LIN {X 0,Y 410.932,Z 415.987,A -85,B 0,C 180,E1 -10557.501,E2 -10557.501} C_VEL
LIN {X 0,Y 411.272,Z 410.477,A -85,B 0,C 180,E1 -10560.841,E2 -10560.841} C_VEL
LIN {X 0,Y 411.519,Z 406.698,A -85,B 0,C 180,E1 -10563.193,E2 -10563.193} C_VEL
LIN {X 0,Y 411.867,Z 401.28,A -85,B 0,C 180,E1 -10566.679,E2 -10566.679} C_VEL
LIN {X 0,Y 411.907,Z 397.623,A -85,B 0,C 180,E1 -10569.146,E2 -10569.146} C_VEL
LIN {X 0,Y 411.508,Z 393.953,A -85,B 0,C 180,E1 -10571.764,E2 -10571.764} C_VEL
LIN {X 0,Y 411.201,Z 391.892,A -85,B 0,C 180,E1 -10573.298,E2 -10573.298} C_VEL
LIN {X 0,Y 411.178,Z 391.895,A -85,B 0,C 180,E1 -10576.867,E2 -10576.867} C_VEL
LIN {X 0,Y 411.229,Z 391.886,A -85,B 0,C 180,E1 -10580.27,E2 -10580.27} C_VEL
LIN {X 0,Y 411.197,Z 391.89,A -85,B 0,C 180,E1 -10583.447,E2 -10583.447} C_VEL
LIN {X 0,Y 411.208,Z 391.889,A -85,B 0,C 180,E1 -10586.873,E2 -10586.873} C_VEL
LIN {X 0,Y 411.234,Z 391.888,A -85,B 0,C 180,E1 -10590.644,E2 -10590.644} C_VEL
LIN {X 0,Y 411.238,Z 391.885,A -85,B 0,C 180,E1 -10593.619,E2 -10593.619} C_VEL
LIN {X 0,Y 411.197,Z 391.89,A -85,B 0,C 180,E1 -10596.852,E2 -10596.852} C_VEL
LIN {X 0,Y 411.216,Z 391.887,A -85,B 0,C 180,E1 -10600.05,E2 -10600.05} C_VEL
LIN {X 0,Y 411.266,Z 391.879,A -85,B 0,C 180,E1 -10603.13,E2 -10603.13} C_VEL
LIN {X 0,Y 411.258,Z 391.88,A -85,B 0,C 180,E1 -10606.158,E2 -10606.158} C_VEL
LIN {X 0,Y 411.289,Z 391.876,A -85,B 0,C 180,E1 -10609.166,E2 -10609.166} C_VEL
LIN {X 0,Y 411.483,Z 391.852,A -85,B 0,C 180,E1 -10612.147,E2 -10612.147} C_VEL
LIN {X 0,Y 411.477,Z 391.854,A -85,B 0,C 180,E1 -10614.118,E2 -10614.118} C_VEL
LIN {X 0,Y 411.516,Z 391.85,A -85,B 0,C 180,E1 -10618.043,E2 -10618.043} C_VEL
LIN {X 0,Y 411.644,Z 391.836,A -85,B 0,C 180,E1 -10620,E2 -10620} C_VEL
LIN {X 0,Y 411.459,Z 391.857,A -85,B 0,C 180,E1 -10622.937,E2 -10622.937} C_VEL
LIN {X 0,Y 411.463,Z 391.857,A -85,B 0,C 180,E1 -10626.867,E2 -10626.867} C_VEL
LIN {X 0,Y 411.306,Z 391.878,A -85,B 0,C 180,E1 -10629.839,E2 -10629.839} C_VEL
LIN {X 0,Y 411.307,Z 391.875,A -85,B 0,C 180,E1 -10633.104,E2 -10633.104} C_VEL
LIN {X 0,Y 411.265,Z 391.882,A -85,B 0,C 180,E1 -10635.868,E2 -10635.868} C_VEL
LIN {X 0,Y 411.227,Z 391.885,A -85,B 0,C 180,E1 -10638.949,E2 -10638.949} C_VEL
LIN {X 0,Y 411.206,Z 391.891,A -85,B 0,C 180,E1 -10642.643,E2 -10642.643} C_VEL
LIN {X 0,Y 411.238,Z 391.884,A -85,B 0,C 180,E1 -10645.293,E2 -10645.293} C_VEL
LIN {X 0,Y 411.26,Z 391.884,A -85,B 0,C 180,E1 -10647.478,E2 -10647.478} C_VEL
LIN {X 0,Y 411.191,Z 391.893,A -85,B 0,C 180,E1 -10650.848,E2 -10650.848} C_VEL
LIN {X 0,Y 411.208,Z 391.89,A -85,B 0,C 180,E1 -10654.333,E2 -10654.333} C_VEL
LIN {X 0,Y 411.202,Z 391.887,A -85,B 0,C 180,E1 -10657.973,E2 -10657.973} C_VEL
LIN {X 0,Y 411.183,Z 391.894,A -85,B 0,C 180,E1 -10660.504,E2 -10660.504} C_VEL
LIN {X 0,Y 411.175,Z 391.893,A -85,B 0,C 180,E1 -10663.134,E2 -10663.134} C_VEL
LIN {X 0,Y 411.175,Z 391.894,A -85,B 0,C 180,E1 -10665.88,E2 -10665.88} C_VEL
LIN {X 0,Y 411.196,Z 392.038,A -85,B 0,C 180,E1 -10668.767,E2 -10668.767} C_VEL
LIN {X 0,Y 411.452,Z 394.537,A -85,B 0,C 180,E1 -10670.803,E2 -10670.803} C_VEL
LIN {X 0,Y 411.471,Z 397.876,A -85,B 0,C 180,E1 -10673.396,E2 -10673.396} C_VEL
LIN {X 0,Y 411.254,Z 402.544,A -85,B 0,C 180,E1 -10676.864,E2 -10676.864} C_VEL
LIN {X 0,Y 411.071,Z 405.713,A -85,B 0,C 180,E1 -10679.143,E2 -10679.143} C_VEL
LIN {X 0,Y 410.798,Z 410.981,A -85,B 0,C 180,E1 -10682.827,E2 -10682.827} C_VEL
LIN {X 0,Y 410.582,Z 415.248,A -85,B 0,C 180,E1 -10685.744,E2 -10685.744} C_VEL
LIN {X 0,Y 410.457,Z 419.829,A -85,B 0,C 180,E1 -10688.754,E2 -10688.754} C_VEL
LIN {X 0,Y 414.185,Z 433.819,A -85,B 0,C 180,E1 -10689.343,E2 -10689.343} C_VEL
LIN {X 0,Y 417.104,Z 447.077,A -85,B 0,C 180,E1 -10690.05,E2 -10690.05} C_VEL
LIN {X 0,Y 417.637,Z 450.91,A -85,B 0,C 180,E1 -10690.269,E2 -10690.269} C_VEL
LIN {X 0,Y 416.849,Z 464.097,A -85,B 0,C 180,E1 -10691.04,E2 -10691.04} C_VEL
LIN {X 0,Y 415.977,Z 475.884,A -85,B 0,C 180,E1 -10691.914,E2 -10691.914} C_VEL
LIN {X 0,Y 414.892,Z 487.847,A -85,B 0,C 180,E1 -10693.01,E2 -10693.01} C_VEL
LIN {X 0,Y 413.863,Z 498.759,A -85,B 0,C 180,E1 -10694.234,E2 -10694.234} C_VEL
LIN {X 0,Y 412.988,Z 508.063,A -85,B 0,C 180,E1 -10695.488,E2 -10695.488} C_VEL
LIN {X 0,Y 412.212,Z 517.264,A -85,B 0,C 180,E1 -10696.983,E2 -10696.983} C_VEL
LIN {X 0,Y 411.336,Z 525.8,A -85,B 0,C 180,E1 -10698.669,E2 -10698.669} C_VEL
LIN {X 0,Y 410.849,Z 531.96,A -85,B 0,C 180,E1 -10700.151,E2 -10700.151} C_VEL
LIN {X 0,Y 410.369,Z 538.494,A -85,B 0,C 180,E1 -10702.125,E2 -10702.125} C_VEL
LIN {X 0,Y 410.135,Z 543.392,A -85,B 0,C 180,E1 -10704.099,E2 -10704.099} C_VEL
LIN {X 0,Y 409.939,Z 546.804,A -85,B 0,C 180,E1 -10706.068,E2 -10706.068} C_VEL
LIN {X 0,Y 409.966,Z 548.829,A -85,B 0,C 180,E1 -10708.035,E2 -10708.035} C_VEL
LIN {X 0,Y 409.905,Z 549.526,A -85,B 0,C 180,E1 -10710,E2 -10710} C_VEL
LIN {X 0,Y 409.966,Z 548.9,A -85,B 0,C 180,E1 -10711.965,E2 -10711.965} C_VEL
LIN {X 0,Y 409.938,Z 546.938,A -85,B 0,C 180,E1 -10713.932,E2 -10713.932} C_VEL
LIN {X 0,Y 410.122,Z 543.591,A -85,B 0,C 180,E1 -10715.902,E2 -10715.902} C_VEL
LIN {X 0,Y 410.365,Z 538.765,A -85,B 0,C 180,E1 -10717.875,E2 -10717.875} C_VEL
LIN {X 0,Y 410.488,Z 536.976,A -85,B 0,C 180,E1 -10718.482,E2 -10718.482} C_VEL
LIN {X 0,Y 409.995,Z 534.605,A -85,B 0,C 180,E1 -10719.231,E2 -10719.231} C_VEL
LIN {X 0,Y 407.5,Z 530.401,A -85,B 0,C 180,E1 -10720.443,E2 -10720.443} C_VEL
LIN {X 0,Y 405.098,Z 525.759,A -85,B 0,C 180,E1 -10721.632,E2 -10721.632} C_VEL
LIN {X 0,Y 404.756,Z 522.548,A -85,B 0,C 180,E1 -10722.334,E2 -10722.334} C_VEL
LIN {X 0,Y 405.592,Z 513.315,A -85,B 0,C 180,E1 -10724.04,E2 -10724.04} C_VEL
LIN {X 0,Y 406.577,Z 503.364,A -85,B 0,C 180,E1 -10725.541,E2 -10725.541} C_VEL
LIN {X 0,Y 407.689,Z 492.287,A -85,B 0,C 180,E1 -10726.912,E2 -10726.912} C_VEL
LIN {X 0,Y 408.768,Z 481.257,A -85,B 0,C 180,E1 -10728.028,E2 -10728.028} C_VEL
LIN {X 0,Y 409.79,Z 469.285,A -85,B 0,C 180,E1 -10729.018,E2 -10729.018} C_VEL
LIN {X 0,Y 410.684,Z 456.556,A -85,B 0,C 180,E1 -10729.855,E2 -10729.855} C_VEL
LIN {X 0,Y 410.884,Z 450.89,A -85,B 0,C 180,E1 -10730.172,E2 -10730.172} C_VEL
LIN {X 0,Y 407.936,Z 436.771,A -85,B 0,C 180,E1 -10730.982,E2 -10730.982} C_VEL
LIN {X 0,Y 404.018,Z 422.414,A -85,B 0,C 180,E1 -10731.644,E2 -10731.644} C_VEL
LIN {X 0,Y 403.384,Z 419.805,A -85,B 0,C 180,E1 -10731.747,E2 -10731.747} C_VEL
LIN {X 0,Y 403.588,Z 414.887,A -85,B 0,C 180,E1 -10735.107,E2 -10735.107} C_VEL
LIN {X 0,Y 403.764,Z 410.679,A -85,B 0,C 180,E1 -10738.032,E2 -10738.032} C_VEL
LIN {X 0,Y 404.09,Z 405.774,A -85,B 0,C 180,E1 -10741.546,E2 -10741.546} C_VEL
LIN {X 0,Y 404.322,Z 401.114,A -85,B 0,C 180,E1 -10745.003,E2 -10745.003} C_VEL
LIN {X 0,Y 404.462,Z 397.921,A -85,B 0,C 180,E1 -10747.457,E2 -10747.457} C_VEL
LIN {X 0,Y 404.367,Z 394.599,A -85,B 0,C 180,E1 -10750.117,E2 -10750.117} C_VEL
LIN {X 0,Y 404.167,Z 392.814,A -85,B 0,C 180,E1 -10751.606,E2 -10751.606} C_VEL
LIN {X 0,Y 404.151,Z 392.773,A -85,B 0,C 180,E1 -10754.523,E2 -10754.523} C_VEL
LIN {X 0,Y 404.139,Z 392.772,A -85,B 0,C 180,E1 -10757.296,E2 -10757.296} C_VEL
LIN {X 0,Y 404.171,Z 392.766,A -85,B 0,C 180,E1 -10759.955,E2 -10759.955} C_VEL
LIN {X 0,Y 404.143,Z 392.769,A -85,B 0,C 180,E1 -10763.124,E2 -10763.124} C_VEL
LIN {X 0,Y 404.148,Z 392.77,A -85,B 0,C 180,E1 -10766.188,E2 -10766.188} C_VEL
LIN {X 0,Y 404.148,Z 392.767,A -85,B 0,C 180,E1 -10769.715,E2 -10769.715} C_VEL
LIN {X 0,Y 404.198,Z 392.761,A -85,B 0,C 180,E1 -10773.123,E2 -10773.123} C_VEL
LIN {X 0,Y 404.18,Z 392.764,A -85,B 0,C 180,E1 -10775.334,E2 -10775.334} C_VEL
LIN {X 0,Y 404.142,Z 392.769,A -85,B 0,C 180,E1 -10778.581,E2 -10778.581} C_VEL
LIN {X 0,Y 404.213,Z 392.76,A -85,B 0,C 180,E1 -10781.762,E2 -10781.762} C_VEL
LIN {X 0,Y 404.21,Z 392.759,A -85,B 0,C 180,E1 -10784.882,E2 -10784.882} C_VEL
LIN {X 0,Y 404.26,Z 392.753,A -85,B 0,C 180,E1 -10787.958,E2 -10787.958} C_VEL
LIN {X 0,Y 404.436,Z 392.734,A -85,B 0,C 180,E1 -10792.1,E2 -10792.1} C_VEL
LIN {X 0,Y 404.427,Z 392.733,A -85,B 0,C 180,E1 -10794.015,E2 -10794.015} C_VEL
LIN {X 0,Y 404.483,Z 392.726,A -85,B 0,C 180,E1 -10798.008,E2 -10798.008} C_VEL
LIN {X 0,Y 404.613,Z 392.713,A -85,B 0,C 180,E1 -10800,E2 -10800} C_VEL
LIN {X 0,Y 404.425,Z 392.734,A -85,B 0,C 180,E1 -10802.988,E2 -10802.988} C_VEL
LIN {X 0,Y 404.415,Z 392.734,A -85,B 0,C 180,E1 -10806.987,E2 -10806.987} C_VEL
LIN {X 0,Y 404.269,Z 392.753,A -85,B 0,C 180,E1 -10810.011,E2 -10810.011} C_VEL
LIN {X 0,Y 404.269,Z 392.755,A -85,B 0,C 180,E1 -10813.211,E2 -10813.211} C_VEL
LIN {X 0,Y 404.218,Z 392.757,A -85,B 0,C 180,E1 -10817.007,E2 -10817.007} C_VEL
LIN {X 0,Y 404.166,Z 392.765,A -85,B 0,C 180,E1 -10820.351,E2 -10820.351} C_VEL
LIN {X 0,Y 404.172,Z 392.761,A -85,B 0,C 180,E1 -10823.574,E2 -10823.574} C_VEL
LIN {X 0,Y 404.186,Z 392.764,A -85,B 0,C 180,E1 -10825.766,E2 -10825.766} C_VEL
LIN {X 0,Y 404.197,Z 392.762,A -85,B 0,C 180,E1 -10827.999,E2 -10827.999} C_VEL
LIN {X 0,Y 404.141,Z 392.768,A -85,B 0,C 180,E1 -10831.558,E2 -10831.558} C_VEL
LIN {X 0,Y 404.188,Z 392.763,A -85,B 0,C 180,E1 -10835.016,E2 -10835.016} C_VEL
LIN {X 0,Y 404.166,Z 392.77,A -85,B 0,C 180,E1 -10838.756,E2 -10838.756} C_VEL
LIN {X 0,Y 404.152,Z 392.77,A -85,B 0,C 180,E1 -10841.604,E2 -10841.604} C_VEL
LIN {X 0,Y 404.147,Z 392.769,A -85,B 0,C 180,E1 -10844.522,E2 -10844.522} C_VEL
LIN {X 0,Y 404.136,Z 392.807,A -85,B 0,C 180,E1 -10846.454,E2 -10846.454} C_VEL
LIN {X 0,Y 404.641,Z 395.775,A -85,B 0,C 180,E1 -10848.7,E2 -10848.7} C_VEL
LIN {X 0,Y 404.907,Z 399.477,A -85,B 0,C 180,E1 -10851.359,E2 -10851.359} C_VEL
LIN {X 0,Y 404.78,Z 403.102,A -85,B 0,C 180,E1 -10853.82,E2 -10853.82} C_VEL
LIN {X 0,Y 404.389,Z 408.592,A -85,B 0,C 180,E1 -10857.401,E2 -10857.401} C_VEL
LIN {X 0,Y 404.057,Z 414.115,A -85,B 0,C 180,E1 -10860.855,E2 -10860.855} C_VEL
LIN {X 0,Y 403.843,Z 417.797,A -85,B 0,C 180,E1 -10863.097,E2 -10863.097} C_VEL
LIN {X 0,Y 403.539,Z 423.318,A -85,B 0,C 180,E1 -10866.386,E2 -10866.386} C_VEL
LIN {X 0,Y 403.447,Z 426.603,A -85,B 0,C 180,E1 -10868.3,E2 -10868.3} C_VEL
LIN {X 0,Y 407.112,Z 441.134,A -85,B 0,C 180,E1 -10868.91,E2 -10868.91} C_VEL
LIN {X 0,Y 409.79,Z 453.958,A -85,B 0,C 180,E1 -10869.593,E2 -10869.593} C_VEL
LIN {X 0,Y 410.664,Z 460.503,A -85,B 0,C 180,E1 -10869.984,E2 -10869.984} C_VEL
LIN {X 0,Y 409.806,Z 474.005,A -85,B 0,C 180,E1 -10870.822,E2 -10870.822} C_VEL
LIN {X 0,Y 408.723,Z 486.899,A -85,B 0,C 180,E1 -10871.841,E2 -10871.841} C_VEL
LIN {X 0,Y 407.496,Z 499.461,A -85,B 0,C 180,E1 -10873.08,E2 -10873.08} C_VEL
LIN {X 0,Y 406.404,Z 510.651,A -85,B 0,C 180,E1 -10874.452,E2 -10874.452} C_VEL
LIN {X 0,Y 405.407,Z 520.686,A -85,B 0,C 180,E1 -10875.954,E2 -10875.954} C_VEL
LIN {X 0,Y 404.707,Z 529.022,A -85,B 0,C 180,E1 -10877.463,E2 -10877.463} C_VEL
LIN {X 0,Y 403.888,Z 536.989,A -85,B 0,C 180,E1 -10879.219,E2 -10879.219} C_VEL
LIN {X 0,Y 403.433,Z 543.405,A -85,B 0,C 180,E1 -10880.98,E2 -10880.98} C_VEL
LIN {X 0,Y 403.072,Z 549.091,A -85,B 0,C 180,E1 -10882.989,E2 -10882.989} C_VEL
LIN {X 0,Y 402.914,Z 553.217,A -85,B 0,C 180,E1 -10884.997,E2 -10884.997} C_VEL
LIN {X 0,Y 402.779,Z 555.911,A -85,B 0,C 180,E1 -10886.999,E2 -10886.999} C_VEL
LIN {X 0,Y 402.843,Z 557.247,A -85,B 0,C 180,E1 -10889,E2 -10889} C_VEL
LIN {X 0,Y 402.843,Z 557.246,A -85,B 0,C 180,E1 -10891,E2 -10891} C_VEL
LIN {X 0,Y 402.779,Z 555.909,A -85,B 0,C 180,E1 -10893.001,E2 -10893.001} C_VEL
LIN {X 0,Y 402.918,Z 553.214,A -85,B 0,C 180,E1 -10895.003,E2 -10895.003} C_VEL
LIN {X 0,Y 403.077,Z 549.081,A -85,B 0,C 180,E1 -10897.01,E2 -10897.01} C_VEL
LIN {X 0,Y 403.418,Z 543.388,A -85,B 0,C 180,E1 -10899.021,E2 -10899.021} C_VEL
LIN {X 0,Y 403.888,Z 536.97,A -85,B 0,C 180,E1 -10900.781,E2 -10900.781} C_VEL
LIN {X 0,Y 404.707,Z 528.998,A -85,B 0,C 180,E1 -10902.537,E2 -10902.537} C_VEL
LIN {X 0,Y 405.409,Z 520.656,A -85,B 0,C 180,E1 -10904.046,E2 -10904.046} C_VEL
LIN {X 0,Y 406.395,Z 510.613,A -85,B 0,C 180,E1 -10905.548,E2 -10905.548} C_VEL
LIN {X 0,Y 407.534,Z 499.41,A -85,B 0,C 180,E1 -10906.919,E2 -10906.919} C_VEL
LIN {X 0,Y 408.742,Z 486.838,A -85,B 0,C 180,E1 -10908.158,E2 -10908.158} C_VEL
LIN {X 0,Y 409.746,Z 474.198,A -85,B 0,C 180,E1 -10909.161,E2 -10909.161} C_VEL
LIN {X 0,Y 410.658,Z 460.385,A -85,B 0,C 180,E1 -10910.016,E2 -10910.016} C_VEL
LIN {X 0,Y 408.735,Z 448.556,A -85,B 0,C 180,E1 -10910.704,E2 -10910.704} C_VEL
LIN {X 0,Y 405.445,Z 434.421,A -85,B 0,C 180,E1 -10911.388,E2 -10911.388} C_VEL
LIN {X 0,Y 403.425,Z 426.53,A -85,B 0,C 180,E1 -10911.727,E2 -10911.727} C_VEL
LIN {X 0,Y 403.646,Z 420.745,A -85,B 0,C 180,E1 -10915.125,E2 -10915.125} C_VEL
LIN {X 0,Y 403.928,Z 415.947,A -85,B 0,C 180,E1 -10918.02,E2 -10918.02} C_VEL
LIN {X 0,Y 404.295,Z 410.171,A -85,B 0,C 180,E1 -10921.594,E2 -10921.594} C_VEL
LIN {X 0,Y 404.632,Z 404.91,A -85,B 0,C 180,E1 -10924.972,E2 -10924.972} C_VEL
LIN {X 0,Y 404.882,Z 401.238,A -85,B 0,C 180,E1 -10927.411,E2 -10927.411} C_VEL
LIN {X 0,Y 404.82,Z 397.26,A -85,B 0,C 180,E1 -10930.193,E2 -10930.193} C_VEL
LIN {X 0,Y 404.258,Z 393.357,A -85,B 0,C 180,E1 -10933.1,E2 -10933.1} C_VEL
LIN {X 0,Y 404.135,Z 392.772,A -85,B 0,C 180,E1 -10933.678,E2 -10933.678} C_VEL
LIN {X 0,Y 404.172,Z 392.768,A -85,B 0,C 180,E1 -10937.3,E2 -10937.3} C_VEL
LIN {X 0,Y 404.169,Z 392.767,A -85,B 0,C 180,E1 -10939.955,E2 -10939.955} C_VEL
LIN {X 0,Y 404.142,Z 392.77,A -85,B 0,C 180,E1 -10943.124,E2 -10943.124} C_VEL
LIN {X 0,Y 404.146,Z 392.771,A -85,B 0,C 180,E1 -10946.188,E2 -10946.188} C_VEL
LIN {X 0,Y 404.146,Z 392.769,A -85,B 0,C 180,E1 -10949.715,E2 -10949.715} C_VEL
LIN {X 0,Y 404.196,Z 392.761,A -85,B 0,C 180,E1 -10953.123,E2 -10953.123} C_VEL
LIN {X 0,Y 404.175,Z 392.765,A -85,B 0,C 180,E1 -10955.334,E2 -10955.334} C_VEL
LIN {X 0,Y 404.139,Z 392.769,A -85,B 0,C 180,E1 -10958.581,E2 -10958.581} C_VEL
LIN {X 0,Y 404.212,Z 392.759,A -85,B 0,C 180,E1 -10961.762,E2 -10961.762} C_VEL
LIN {X 0,Y 404.214,Z 392.759,A -85,B 0,C 180,E1 -10964.882,E2 -10964.882} C_VEL
LIN {X 0,Y 404.258,Z 392.753,A -85,B 0,C 180,E1 -10967.959,E2 -10967.959} C_VEL
LIN {X 0,Y 404.435,Z 392.73,A -85,B 0,C 180,E1 -10972.1,E2 -10972.1} C_VEL
LIN {X 0,Y 404.426,Z 392.733,A -85,B 0,C 180,E1 -10974.015,E2 -10974.015} C_VEL
LIN {X 0,Y 404.485,Z 392.726,A -85,B 0,C 180,E1 -10978.009,E2 -10978.009} C_VEL
LIN {X 0,Y 404.613,Z 392.712,A -85,B 0,C 180,E1 -10980,E2 -10980} C_VEL
LIN {X 0,Y 404.418,Z 392.734,A -85,B 0,C 180,E1 -10982.989,E2 -10982.989} C_VEL
LIN {X 0,Y 404.414,Z 392.734,A -85,B 0,C 180,E1 -10986.987,E2 -10986.987} C_VEL
LIN {X 0,Y 404.268,Z 392.753,A -85,B 0,C 180,E1 -10990.012,E2 -10990.012} C_VEL
LIN {X 0,Y 404.268,Z 392.751,A -85,B 0,C 180,E1 -10993.211,E2 -10993.211} C_VEL
LIN {X 0,Y 404.221,Z 392.755,A -85,B 0,C 180,E1 -10997.009,E2 -10997.009} C_VEL
LIN {X 0,Y 404.165,Z 392.764,A -85,B 0,C 180,E1 -11000.352,E2 -11000.352} C_VEL
LIN {X 0,Y 404.171,Z 392.764,A -85,B 0,C 180,E1 -11003.575,E2 -11003.575} C_VEL
LIN {X 0,Y 404.185,Z 392.765,A -85,B 0,C 180,E1 -11005.766,E2 -11005.766} C_VEL
LIN {X 0,Y 404.197,Z 392.762,A -85,B 0,C 180,E1 -11008,E2 -11008} C_VEL
LIN {X 0,Y 404.14,Z 392.768,A -85,B 0,C 180,E1 -11011.558,E2 -11011.558} C_VEL
LIN {X 0,Y 404.187,Z 392.762,A -85,B 0,C 180,E1 -11015.016,E2 -11015.016} C_VEL
LIN {X 0,Y 404.16,Z 392.767,A -85,B 0,C 180,E1 -11018.757,E2 -11018.757} C_VEL
LIN {X 0,Y 404.124,Z 392.77,A -85,B 0,C 180,E1 -11021.6,E2 -11021.6} C_VEL
LIN {X 0,Y 404.148,Z 392.768,A -85,B 0,C 180,E1 -11024.522,E2 -11024.522} C_VEL
LIN {X 0,Y 404.142,Z 392.771,A -85,B 0,C 180,E1 -11027.296,E2 -11027.296} C_VEL
LIN {X 0,Y 404.16,Z 392.979,A -85,B 0,C 180,E1 -11028.64,E2 -11028.64} C_VEL
LIN {X 0,Y 404.451,Z 396.387,A -85,B 0,C 180,E1 -11031.44,E2 -11031.44} C_VEL
LIN {X 0,Y 404.391,Z 399.375,A -85,B 0,C 180,E1 -11033.78,E2 -11033.78} C_VEL
LIN {X 0,Y 404.218,Z 403.085,A -85,B 0,C 180,E1 -11036.57,E2 -11036.57} C_VEL
LIN {X 0,Y 403.939,Z 407.362,A -85,B 0,C 180,E1 -11039.698,E2 -11039.698} C_VEL
LIN {X 0,Y 403.73,Z 412.128,A -85,B 0,C 180,E1 -11043.089,E2 -11043.089} C_VEL
LIN {X 0,Y 403.48,Z 416.909,A -85,B 0,C 180,E1 -11046.383,E2 -11046.383} C_VEL
LIN {X 0,Y 403.416,Z 419.809,A -85,B 0,C 180,E1 -11048.356,E2 -11048.356} C_VEL
LIN {X 0,Y 407.494,Z 435.085,A -85,B 0,C 180,E1 -11049.031,E2 -11049.031} C_VEL
LIN {X 0,Y 410.403,Z 448.443,A -85,B 0,C 180,E1 -11049.775,E2 -11049.775} C_VEL
LIN {X 0,Y 410.898,Z 452.117,A -85,B 0,C 180,E1 -11049.996,E2 -11049.996} C_VEL
LIN {X 0,Y 410.111,Z 464.554,A -85,B 0,C 180,E1 -11050.745,E2 -11050.745} C_VEL
LIN {X 0,Y 409.097,Z 477.382,A -85,B 0,C 180,E1 -11051.728,E2 -11051.728} C_VEL
LIN {X 0,Y 407.826,Z 490.264,A -85,B 0,C 180,E1 -11052.965,E2 -11052.965} C_VEL
LIN {X 0,Y 406.808,Z 500.78,A -85,B 0,C 180,E1 -11054.211,E2 -11054.211} C_VEL
LIN {X 0,Y 405.763,Z 511.22,A -85,B 0,C 180,E1 -11055.711,E2 -11055.711} C_VEL
LIN {X 0,Y 405.038,Z 519.829,A -85,B 0,C 180,E1 -11057.219,E2 -11057.219} C_VEL
LIN {X 0,Y 404.144,Z 528.084,A -85,B 0,C 180,E1 -11058.972,E2 -11058.972} C_VEL
LIN {X 0,Y 403.669,Z 533.835,A -85,B 0,C 180,E1 -11060.48,E2 -11060.48} C_VEL
LIN {X 0,Y 403.309,Z 538.564,A -85,B 0,C 180,E1 -11061.987,E2 -11061.987} C_VEL
LIN {X 0,Y 403.061,Z 543.462,A -85,B 0,C 180,E1 -11063.995,E2 -11063.995} C_VEL
LIN {X 0,Y 402.862,Z 546.873,A -85,B 0,C 180,E1 -11065.999,E2 -11065.999} C_VEL
LIN {X 0,Y 402.864,Z 548.899,A -85,B 0,C 180,E1 -11068.001,E2 -11068.001} C_VEL
LIN {X 0,Y 402.831,Z 549.595,A -85,B 0,C 180,E1 -11070,E2 -11070} C_VEL
LIN {X 0,Y 402.863,Z 548.968,A -85,B 0,C 180,E1 -11072,E2 -11072} C_VEL
LIN {X 0,Y 402.861,Z 547.006,A -85,B 0,C 180,E1 -11074.002,E2 -11074.002} C_VEL
LIN {X 0,Y 403.066,Z 543.659,A -85,B 0,C 180,E1 -11076.005,E2 -11076.005} C_VEL
LIN {X 0,Y 403.305,Z 538.833,A -85,B 0,C 180,E1 -11078.014,E2 -11078.014} C_VEL
LIN {X 0,Y 403.812,Z 532.37,A -85,B 0,C 180,E1 -11080.023,E2 -11080.023} C_VEL
LIN {X 0,Y 404.482,Z 525.173,A -85,B 0,C 180,E1 -11081.78,E2 -11081.78} C_VEL
LIN {X 0,Y 404.756,Z 522.548,A -85,B 0,C 180,E1 -11082.334,E2 -11082.334} C_VEL
LIN {X 0,Y 404.417,Z 519.204,A -85,B 0,C 180,E1 -11083.022,E2 -11083.022} C_VEL
LIN {X 0,Y 402.101,Z 513.578,A -85,B 0,C 180,E1 -11084.14,E2 -11084.14} C_VEL
LIN {X 0,Y 399.893,Z 507.491,A -85,B 0,C 180,E1 -11085.213,E2 -11085.213} C_VEL
LIN {X 0,Y 399.716,Z 503.39,A -85,B 0,C 180,E1 -11085.821,E2 -11085.821} C_VEL
LIN {X 0,Y 400.882,Z 492.352,A -85,B 0,C 180,E1 -11087.208,E2 -11087.208} C_VEL
LIN {X 0,Y 402.01,Z 481.321,A -85,B 0,C 180,E1 -11088.342,E2 -11088.342} C_VEL
LIN {X 0,Y 403.143,Z 468.201,A -85,B 0,C 180,E1 -11089.43,E2 -11089.43} C_VEL
LIN {X 0,Y 404.062,Z 455.371,A -85,B 0,C 180,E1 -11090.268,E2 -11090.268} C_VEL
LIN {X 0,Y 404.018,Z 451.377,A -85,B 0,C 180,E1 -11090.506,E2 -11090.506} C_VEL
LIN {X 0,Y 401.064,Z 437.305,A -85,B 0,C 180,E1 -11091.341,E2 -11091.341} C_VEL
LIN {X 0,Y 397.142,Z 422.944,A -85,B 0,C 180,E1 -11092.027,E2 -11092.027} C_VEL
LIN {X 0,Y 396.32,Z 419.873,A -85,B 0,C 180,E1 -11092.158,E2 -11092.158} C_VEL
LIN {X 0,Y 396.549,Z 415.296,A -85,B 0,C 180,E1 -11095.328,E2 -11095.328} C_VEL
LIN {X 0,Y 396.739,Z 410.746,A -85,B 0,C 180,E1 -11098.574,E2 -11098.574} C_VEL
LIN {X 0,Y 397.06,Z 405.967,A -85,B 0,C 180,E1 -11102.073,E2 -11102.073} C_VEL
LIN {X 0,Y 397.316,Z 401.388,A -85,B 0,C 180,E1 -11105.543,E2 -11105.543} C_VEL
LIN {X 0,Y 397.436,Z 397.971,A -85,B 0,C 180,E1 -11108.237,E2 -11108.237} C_VEL
LIN {X 0,Y 397.251,Z 394.759,A -85,B 0,C 180,E1 -11110.889,E2 -11110.889} C_VEL
LIN {X 0,Y 397.105,Z 393.648,A -85,B 0,C 180,E1 -11111.985,E2 -11111.985} C_VEL
LIN {X 0,Y 397.092,Z 393.649,A -85,B 0,C 180,E1 -11115.068,E2 -11115.068} C_VEL
LIN {X 0,Y 397.069,Z 393.654,A -85,B 0,C 180,E1 -11118.021,E2 -11118.021} C_VEL
LIN {X 0,Y 397.135,Z 393.644,A -85,B 0,C 180,E1 -11121.138,E2 -11121.138} C_VEL
LIN {X 0,Y 397.123,Z 393.646,A -85,B 0,C 180,E1 -11124.496,E2 -11124.496} C_VEL
LIN {X 0,Y 397.081,Z 393.648,A -85,B 0,C 180,E1 -11127.928,E2 -11127.928} C_VEL
LIN {X 0,Y 397.125,Z 393.642,A -85,B 0,C 180,E1 -11131.456,E2 -11131.456} C_VEL
LIN {X 0,Y 397.156,Z 393.639,A -85,B 0,C 180,E1 -11134.488,E2 -11134.488} C_VEL
LIN {X 0,Y 397.112,Z 393.643,A -85,B 0,C 180,E1 -11137.086,E2 -11137.086} C_VEL
LIN {X 0,Y 397.151,Z 393.637,A -85,B 0,C 180,E1 -11140.353,E2 -11140.353} C_VEL
LIN {X 0,Y 397.17,Z 393.638,A -85,B 0,C 180,E1 -11143.553,E2 -11143.553} C_VEL
LIN {X 0,Y 397.231,Z 393.629,A -85,B 0,C 180,E1 -11146.703,E2 -11146.703} C_VEL
LIN {X 0,Y 397.221,Z 393.63,A -85,B 0,C 180,E1 -11149.809,E2 -11149.809} C_VEL
LIN {X 0,Y 397.367,Z 393.611,A -85,B 0,C 180,E1 -11152.888,E2 -11152.888} C_VEL
LIN {X 0,Y 397.257,Z 393.627,A -85,B 0,C 180,E1 -11154.925,E2 -11154.925} C_VEL
LIN {X 0,Y 397.452,Z 393.602,A -85,B 0,C 180,E1 -11157.973,E2 -11157.973} C_VEL
LIN {X 0,Y 397.582,Z 393.588,A -85,B 0,C 180,E1 -11160,E2 -11160} C_VEL
LIN {X 0,Y 397.384,Z 393.612,A -85,B 0,C 180,E1 -11163.041,E2 -11163.041} C_VEL
LIN {X 0,Y 397.367,Z 393.612,A -85,B 0,C 180,E1 -11167.112,E2 -11167.112} C_VEL
LIN {X 0,Y 397.227,Z 393.629,A -85,B 0,C 180,E1 -11170.191,E2 -11170.191} C_VEL
LIN {X 0,Y 397.229,Z 393.631,A -85,B 0,C 180,E1 -11173.321,E2 -11173.321} C_VEL
LIN {X 0,Y 397.184,Z 393.633,A -85,B 0,C 180,E1 -11177.155,E2 -11177.155} C_VEL
LIN {X 0,Y 397.105,Z 393.646,A -85,B 0,C 180,E1 -11180.73,E2 -11180.73} C_VEL
LIN {X 0,Y 397.136,Z 393.638,A -85,B 0,C 180,E1 -11184.018,E2 -11184.018} C_VEL
LIN {X 0,Y 397.196,Z 393.632,A -85,B 0,C 180,E1 -11187.39,E2 -11187.39} C_VEL
LIN {X 0,Y 397.081,Z 393.65,A -85,B 0,C 180,E1 -11190.882,E2 -11190.882} C_VEL
LIN {X 0,Y 397.128,Z 393.644,A -85,B 0,C 180,E1 -11194.493,E2 -11194.493} C_VEL
LIN {X 0,Y 397.112,Z 393.647,A -85,B 0,C 180,E1 -11198.274,E2 -11198.274} C_VEL
LIN {X 0,Y 397.115,Z 393.647,A -85,B 0,C 180,E1 -11200.905,E2 -11200.905} C_VEL
LIN {X 0,Y 397.104,Z 393.648,A -85,B 0,C 180,E1 -11203.648,E2 -11203.648} C_VEL
LIN {X 0,Y 397.108,Z 393.668,A -85,B 0,C 180,E1 -11206.177,E2 -11206.177} C_VEL
LIN {X 0,Y 397.693,Z 397.56,A -85,B 0,C 180,E1 -11209.166,E2 -11209.166} C_VEL
LIN {X 0,Y 397.871,Z 401.218,A -85,B 0,C 180,E1 -11211.812,E2 -11211.812} C_VEL
LIN {X 0,Y 397.685,Z 404.966,A -85,B 0,C 180,E1 -11214.383,E2 -11214.383} C_VEL
LIN {X 0,Y 397.294,Z 410.374,A -85,B 0,C 180,E1 -11217.948,E2 -11217.948} C_VEL
LIN {X 0,Y 396.931,Z 415.89,A -85,B 0,C 180,E1 -11221.441,E2 -11221.441} C_VEL
LIN {X 0,Y 396.608,Z 421.131,A -85,B 0,C 180,E1 -11224.653,E2 -11224.653} C_VEL
LIN {X 0,Y 396.394,Z 426.516,A -85,B 0,C 180,E1 -11227.892,E2 -11227.892} C_VEL
LIN {X 0,Y 400.219,Z 441.498,A -85,B 0,C 180,E1 -11228.544,E2 -11228.544} C_VEL
LIN {X 0,Y 403.125,Z 455.373,A -85,B 0,C 180,E1 -11229.316,E2 -11229.316} C_VEL
LIN {X 0,Y 403.905,Z 460.439,A -85,B 0,C 180,E1 -11229.635,E2 -11229.635} C_VEL
LIN {X 0,Y 403.22,Z 472.633,A -85,B 0,C 180,E1 -11230.398,E2 -11230.398} C_VEL
LIN {X 0,Y 402.068,Z 485.407,A -85,B 0,C 180,E1 -11231.397,E2 -11231.397} C_VEL
LIN {X 0,Y 400.919,Z 497.047,A -85,B 0,C 180,E1 -11232.53,E2 -11232.53} C_VEL
LIN {X 0,Y 399.938,Z 506.736,A -85,B 0,C 180,E1 -11233.67,E2 -11233.67} C_VEL
LIN {X 0,Y 398.777,Z 517.469,A -85,B 0,C 180,E1 -11235.194,E2 -11235.194} C_VEL
LIN {X 0,Y 397.905,Z 526.332,A -85,B 0,C 180,E1 -11236.726,E2 -11236.726} C_VEL
LIN {X 0,Y 397.254,Z 533.707,A -85,B 0,C 180,E1 -11238.261,E2 -11238.261} C_VEL
LIN {X 0,Y 396.679,Z 539.855,A -85,B 0,C 180,E1 -11239.795,E2 -11239.795} C_VEL
LIN {X 0,Y 396.15,Z 546.385,A -85,B 0,C 180,E1 -11241.841,E2 -11241.841} C_VEL
LIN {X 0,Y 395.909,Z 551.272,A -85,B 0,C 180,E1 -11243.886,E2 -11243.886} C_VEL
LIN {X 0,Y 395.754,Z 554.669,A -85,B 0,C 180,E1 -11245.927,E2 -11245.927} C_VEL
LIN {X 0,Y 395.717,Z 556.678,A -85,B 0,C 180,E1 -11247.964,E2 -11247.964} C_VEL
LIN {X 0,Y 395.758,Z 557.344,A -85,B 0,C 180,E1 -11250,E2 -11250} C_VEL
LIN {X 0,Y 395.717,Z 556.676,A -85,B 0,C 180,E1 -11252.035,E2 -11252.035} C_VEL
LIN {X 0,Y 395.755,Z 554.666,A -85,B 0,C 180,E1 -11254.073,E2 -11254.073} C_VEL
LIN {X 0,Y 395.909,Z 551.264,A -85,B 0,C 180,E1 -11256.114,E2 -11256.114} C_VEL
LIN {X 0,Y 396.15,Z 546.368,A -85,B 0,C 180,E1 -11258.159,E2 -11258.159} C_VEL
LIN {X 0,Y 396.678,Z 539.835,A -85,B 0,C 180,E1 -11260.205,E2 -11260.205} C_VEL
LIN {X 0,Y 397.343,Z 532.565,A -85,B 0,C 180,E1 -11261.995,E2 -11261.995} C_VEL
LIN {X 0,Y 398.165,Z 523.994,A -85,B 0,C 180,E1 -11263.707,E2 -11263.707} C_VEL
LIN {X 0,Y 399.133,Z 514.109,A -85,B 0,C 180,E1 -11265.315,E2 -11265.315} C_VEL
LIN {X 0,Y 400.247,Z 503.647,A -85,B 0,C 180,E1 -11266.71,E2 -11266.71} C_VEL
LIN {X 0,Y 401.432,Z 492.101,A -85,B 0,C 180,E1 -11267.973,E2 -11267.973} C_VEL
LIN {X 0,Y 402.622,Z 479.291,A -85,B 0,C 180,E1 -11269.104,E2 -11269.104} C_VEL
LIN {X 0,Y 403.69,Z 465.532,A -85,B 0,C 180,E1 -11270.061,E2 -11270.061} C_VEL
LIN {X 0,Y 403.706,Z 459.176,A -85,B 0,C 180,E1 -11270.442,E2 -11270.442} C_VEL
LIN {X 0,Y 401.095,Z 445.237,A -85,B 0,C 180,E1 -11271.259,E2 -11271.259} C_VEL
LIN {X 0,Y 397.531,Z 431.021,A -85,B 0,C 180,E1 -11271.93,E2 -11271.93} C_VEL
LIN {X 0,Y 396.372,Z 426.475,A -85,B 0,C 180,E1 -11272.125,E2 -11272.125} C_VEL
LIN {X 0,Y 396.603,Z 421.118,A -85,B 0,C 180,E1 -11275.345,E2 -11275.345} C_VEL
LIN {X 0,Y 396.924,Z 415.873,A -85,B 0,C 180,E1 -11278.559,E2 -11278.559} C_VEL
LIN {X 0,Y 397.293,Z 410.354,A -85,B 0,C 180,E1 -11282.052,E2 -11282.052} C_VEL
LIN {X 0,Y 397.684,Z 404.945,A -85,B 0,C 180,E1 -11285.617,E2 -11285.617} C_VEL
LIN {X 0,Y 397.871,Z 401.195,A -85,B 0,C 180,E1 -11288.188,E2 -11288.188} C_VEL
LIN {X 0,Y 397.681,Z 397.534,A -85,B 0,C 180,E1 -11290.835,E2 -11290.835} C_VEL
LIN {X 0,Y 397.086,Z 393.65,A -85,B 0,C 180,E1 -11293.826,E2 -11293.826} C_VEL
LIN {X 0,Y 397.105,Z 393.65,A -85,B 0,C 180,E1 -11296.521,E2 -11296.521} C_VEL
LIN {X 0,Y 397.122,Z 393.646,A -85,B 0,C 180,E1 -11299.551,E2 -11299.551} C_VEL
LIN {X 0,Y 397.101,Z 393.648,A -85,B 0,C 180,E1 -11302.79,E2 -11302.79} C_VEL
LIN {X 0,Y 397.119,Z 393.645,A -85,B 0,C 180,E1 -11306.282,E2 -11306.282} C_VEL
LIN {X 0,Y 397.106,Z 393.645,A -85,B 0,C 180,E1 -11310.135,E2 -11310.135} C_VEL
LIN {X 0,Y 397.195,Z 393.636,A -85,B 0,C 180,E1 -11312.61,E2 -11312.61} C_VEL
LIN {X 0,Y 397.129,Z 393.643,A -85,B 0,C 180,E1 -11315.982,E2 -11315.982} C_VEL
LIN {X 0,Y 397.14,Z 393.639,A -85,B 0,C 180,E1 -11319.705,E2 -11319.705} C_VEL
LIN {X 0,Y 397.185,Z 393.633,A -85,B 0,C 180,E1 -11322.844,E2 -11322.844} C_VEL
LIN {X 0,Y 397.181,Z 393.635,A -85,B 0,C 180,E1 -11325.657,E2 -11325.657} C_VEL
LIN {X 0,Y 397.201,Z 393.632,A -85,B 0,C 180,E1 -11328.777,E2 -11328.777} C_VEL
LIN {X 0,Y 397.396,Z 393.607,A -85,B 0,C 180,E1 -11332.041,E2 -11332.041} C_VEL
LIN {X 0,Y 397.257,Z 393.627,A -85,B 0,C 180,E1 -11334.925,E2 -11334.925} C_VEL
LIN {X 0,Y 397.453,Z 393.601,A -85,B 0,C 180,E1 -11337.973,E2 -11337.973} C_VEL
LIN {X 0,Y 397.583,Z 393.587,A -85,B 0,C 180,E1 -11340,E2 -11340} C_VEL
LIN {X 0,Y 397.377,Z 393.612,A -85,B 0,C 180,E1 -11343.042,E2 -11343.042} C_VEL
LIN {X 0,Y 397.366,Z 393.612,A -85,B 0,C 180,E1 -11347.112,E2 -11347.112} C_VEL
LIN {X 0,Y 397.226,Z 393.629,A -85,B 0,C 180,E1 -11350.191,E2 -11350.191} C_VEL
LIN {X 0,Y 397.228,Z 393.627,A -85,B 0,C 180,E1 -11353.321,E2 -11353.321} C_VEL
LIN {X 0,Y 397.173,Z 393.635,A -85,B 0,C 180,E1 -11356.447,E2 -11356.447} C_VEL
LIN {X 0,Y 397.15,Z 393.641,A -85,B 0,C 180,E1 -11359.647,E2 -11359.647} C_VEL
LIN {X 0,Y 397.137,Z 393.642,A -85,B 0,C 180,E1 -11363.041,E2 -11363.041} C_VEL
LIN {X 0,Y 397.137,Z 393.642,A -85,B 0,C 180,E1 -11366.258,E2 -11366.258} C_VEL
LIN {X 0,Y 397.123,Z 393.642,A -85,B 0,C 180,E1 -11368.544,E2 -11368.544} C_VEL
LIN {X 0,Y 397.08,Z 393.649,A -85,B 0,C 180,E1 -11372.072,E2 -11372.072} C_VEL
LIN {X 0,Y 397.122,Z 393.645,A -85,B 0,C 180,E1 -11375.504,E2 -11375.504} C_VEL
LIN {X 0,Y 397.134,Z 393.643,A -85,B 0,C 180,E1 -11378.862,E2 -11378.862} C_VEL
LIN {X 0,Y 397.07,Z 393.652,A -85,B 0,C 180,E1 -11382.267,E2 -11382.267} C_VEL
LIN {X 0,Y 397.092,Z 393.649,A -85,B 0,C 180,E1 -11385.068,E2 -11385.068} C_VEL
LIN {X 0,Y 397.079,Z 393.65,A -85,B 0,C 180,E1 -11388.019,E2 -11388.019} C_VEL
LIN {X 0,Y 397.354,Z 396.232,A -85,B 0,C 180,E1 -11390.452,E2 -11390.452} C_VEL
LIN {X 0,Y 397.422,Z 399.431,A -85,B 0,C 180,E1 -11393.04,E2 -11393.04} C_VEL
LIN {X 0,Y 397.154,Z 404.223,A -85,B 0,C 180,E1 -11396.731,E2 -11396.731} C_VEL
LIN {X 0,Y 396.954,Z 407.427,A -85,B 0,C 180,E1 -11399.107,E2 -11399.107} C_VEL
LIN {X 0,Y 396.708,Z 412.201,A -85,B 0,C 180,E1 -11402.573,E2 -11402.573} C_VEL
LIN {X 0,Y 396.457,Z 416.972,A -85,B 0,C 180,E1 -11405.938,E2 -11405.938} C_VEL
LIN {X 0,Y 396.387,Z 420.083,A -85,B 0,C 180,E1 -11407.962,E2 -11407.962} C_VEL
LIN {X 0,Y 400.495,Z 435.037,A -85,B 0,C 180,E1 -11408.642,E2 -11408.642} C_VEL
LIN {X 0,Y 403.486,Z 448.536,A -85,B 0,C 180,E1 -11409.413,E2 -11409.413} C_VEL
LIN {X 0,Y 404.129,Z 453.635,A -85,B 0,C 180,E1 -11409.731,E2 -11409.731} C_VEL
LIN {X 0,Y 403.272,Z 466.568,A -85,B 0,C 180,E1 -11410.551,E2 -11410.551} C_VEL
LIN {X 0,Y 402.225,Z 478.88,A -85,B 0,C 180,E1 -11411.537,E2 -11411.537} C_VEL
LIN {X 0,Y 401.05,Z 490.338,A -85,B 0,C 180,E1 -11412.668,E2 -11412.668} C_VEL
LIN {X 0,Y 399.958,Z 500.852,A -85,B 0,C 180,E1 -11413.933,E2 -11413.933} C_VEL
LIN {X 0,Y 398.853,Z 511.292,A -85,B 0,C 180,E1 -11415.458,E2 -11415.458} C_VEL
LIN {X 0,Y 398.079,Z 519.901,A -85,B 0,C 180,E1 -11416.991,E2 -11416.991} C_VEL
LIN {X 0,Y 397.14,Z 528.156,A -85,B 0,C 180,E1 -11418.775,E2 -11418.775} C_VEL
LIN {X 0,Y 396.645,Z 533.906,A -85,B 0,C 180,E1 -11420.31,E2 -11420.31} C_VEL
LIN {X 0,Y 396.25,Z 538.635,A -85,B 0,C 180,E1 -11421.843,E2 -11421.843} C_VEL
LIN {X 0,Y 395.998,Z 543.532,A -85,B 0,C 180,E1 -11423.887,E2 -11423.887} C_VEL
LIN {X 0,Y 395.787,Z 546.943,A -85,B 0,C 180,E1 -11425.927,E2 -11425.927} C_VEL
LIN {X 0,Y 395.762,Z 548.968,A -85,B 0,C 180,E1 -11427.965,E2 -11427.965} C_VEL
LIN {X 0,Y 395.759,Z 549.664,A -85,B 0,C 180,E1 -11430,E2 -11430} C_VEL
LIN {X 0,Y 395.761,Z 549.037,A -85,B 0,C 180,E1 -11432.035,E2 -11432.035} C_VEL
LIN {X 0,Y 395.786,Z 547.074,A -85,B 0,C 180,E1 -11434.073,E2 -11434.073} C_VEL
LIN {X 0,Y 395.998,Z 543.727,A -85,B 0,C 180,E1 -11436.113,E2 -11436.113} C_VEL
LIN {X 0,Y 396.247,Z 538.901,A -85,B 0,C 180,E1 -11438.157,E2 -11438.157} C_VEL
LIN {X 0,Y 396.803,Z 532.438,A -85,B 0,C 180,E1 -11440.202,E2 -11440.202} C_VEL
LIN {X 0,Y 397.519,Z 525.24,A -85,B 0,C 180,E1 -11441.99,E2 -11441.99} C_VEL
LIN {X 0,Y 398.303,Z 517.523,A -85,B 0,C 180,E1 -11443.555,E2 -11443.555} C_VEL
LIN {X 0,Y 399.152,Z 508.643,A -85,B 0,C 180,E1 -11445.053,E2 -11445.053} C_VEL
LIN {X 0,Y 399.716,Z 503.39,A -85,B 0,C 180,E1 -11445.821,E2 -11445.821} C_VEL
LIN {X 0,Y 399.566,Z 499.169,A -85,B 0,C 180,E1 -11446.41,E2 -11446.41} C_VEL
LIN {X 0,Y 397.528,Z 492.166,A -85,B 0,C 180,E1 -11447.385,E2 -11447.385} C_VEL
LIN {X 0,Y 395.527,Z 484.819,A -85,B 0,C 180,E1 -11448.302,E2 -11448.302} C_VEL
LIN {X 0,Y 395.423,Z 479.988,A -85,B 0,C 180,E1 -11448.792,E2 -11448.792} C_VEL
LIN {X 0,Y 396.527,Z 467.445,A -85,B 0,C 180,E1 -11449.831,E2 -11449.831} C_VEL
LIN {X 0,Y 397.481,Z 453.916,A -85,B 0,C 180,E1 -11450.709,E2 -11450.709} C_VEL
LIN {X 0,Y 394.695,Z 439.91,A -85,B 0,C 180,E1 -11451.592,E2 -11451.592} C_VEL
LIN {X 0,Y 390.958,Z 425.875,A -85,B 0,C 180,E1 -11452.318,E2 -11452.318} C_VEL
LIN {X 0,Y 389.273,Z 419.939,A -85,B 0,C 180,E1 -11452.578,E2 -11452.578} C_VEL
LIN {X 0,Y 389.507,Z 415.59,A -85,B 0,C 180,E1 -11455.661,E2 -11455.661} C_VEL
LIN {X 0,Y 389.732,Z 410.812,A -85,B 0,C 180,E1 -11459.136,E2 -11459.136} C_VEL
LIN {X 0,Y 390.049,Z 406.003,A -85,B 0,C 180,E1 -11462.721,E2 -11462.721} C_VEL
LIN {X 0,Y 390.292,Z 401.946,A -85,B 0,C 180,E1 -11465.873,E2 -11465.873} C_VEL
LIN {X 0,Y 390.41,Z 399.622,A -85,B 0,C 180,E1 -11467.738,E2 -11467.738} C_VEL
LIN {X 0,Y 390.267,Z 395.883,A -85,B 0,C 180,E1 -11470.857,E2 -11470.857} C_VEL
LIN {X 0,Y 390.087,Z 394.8,A -85,B 0,C 180,E1 -11471.806,E2 -11471.806} C_VEL
LIN {X 0,Y 390.072,Z 394.525,A -85,B 0,C 180,E1 -11473.209,E2 -11473.209} C_VEL
LIN {X 0,Y 390.06,Z 394.527,A -85,B 0,C 180,E1 -11476.79,E2 -11476.79} C_VEL
LIN {X 0,Y 390.059,Z 394.526,A -85,B 0,C 180,E1 -11479.561,E2 -11479.561} C_VEL
LIN {X 0,Y 390.048,Z 394.524,A -85,B 0,C 180,E1 -11482.449,E2 -11482.449} C_VEL
LIN {X 0,Y 390.087,Z 394.521,A -85,B 0,C 180,E1 -11486.047,E2 -11486.047} C_VEL
LIN {X 0,Y 390.049,Z 394.523,A -85,B 0,C 180,E1 -11489.869,E2 -11489.869} C_VEL
LIN {X 0,Y 390.116,Z 394.515,A -85,B 0,C 180,E1 -11493.232,E2 -11493.232} C_VEL
LIN {X 0,Y 390.109,Z 394.513,A -85,B 0,C 180,E1 -11496.75,E2 -11496.75} C_VEL
LIN {X 0,Y 390.107,Z 394.512,A -85,B 0,C 180,E1 -11499.983,E2 -11499.983} C_VEL
LIN {X 0,Y 390.141,Z 394.512,A -85,B 0,C 180,E1 -11503.248,E2 -11503.248} C_VEL
LIN {X 0,Y 390.197,Z 394.505,A -85,B 0,C 180,E1 -11506.562,E2 -11506.562} C_VEL
LIN {X 0,Y 390.171,Z 394.508,A -85,B 0,C 180,E1 -11509.623,E2 -11509.623} C_VEL
LIN {X 0,Y 390.321,Z 394.489,A -85,B 0,C 180,E1 -11512.759,E2 -11512.759} C_VEL
LIN {X 0,Y 390.229,Z 394.502,A -85,B 0,C 180,E1 -11514.833,E2 -11514.833} C_VEL
LIN {X 0,Y 390.421,Z 394.477,A -85,B 0,C 180,E1 -11517.937,E2 -11517.937} C_VEL
LIN {X 0,Y 390.551,Z 394.464,A -85,B 0,C 180,E1 -11520,E2 -11520} C_VEL
LIN {X 0,Y 390.318,Z 394.492,A -85,B 0,C 180,E1 -11523.096,E2 -11523.096} C_VEL
LIN {X 0,Y 390.333,Z 394.488,A -85,B 0,C 180,E1 -11526.202,E2 -11526.202} C_VEL
LIN {X 0,Y 390.318,Z 394.492,A -85,B 0,C 180,E1 -11528.282,E2 -11528.282} C_VEL
LIN {X 0,Y 390.174,Z 394.508,A -85,B 0,C 180,E1 -11532.483,E2 -11532.483} C_VEL
LIN {X 0,Y 390.142,Z 394.512,A -85,B 0,C 180,E1 -11535.677,E2 -11535.677} C_VEL
LIN {X 0,Y 390.108,Z 394.516,A -85,B 0,C 180,E1 -11538.922,E2 -11538.922} C_VEL
LIN {X 0,Y 390.043,Z 394.525,A -85,B 0,C 180,E1 -11542.234,E2 -11542.234} C_VEL
LIN {X 0,Y 390.122,Z 394.516,A -85,B 0,C 180,E1 -11545.743,E2 -11545.743} C_VEL
LIN {X 0,Y 390.061,Z 394.525,A -85,B 0,C 180,E1 -11549.109,E2 -11549.109} C_VEL
LIN {X 0,Y 390.045,Z 394.527,A -85,B 0,C 180,E1 -11552.721,E2 -11552.721} C_VEL
LIN {X 0,Y 390.06,Z 394.527,A -85,B 0,C 180,E1 -11555.826,E2 -11555.826} C_VEL
LIN {X 0,Y 390.077,Z 394.525,A -85,B 0,C 180,E1 -11559.219,E2 -11559.219} C_VEL
LIN {X 0,Y 390.082,Z 394.523,A -85,B 0,C 180,E1 -11562.38,E2 -11562.38} C_VEL
LIN {X 0,Y 390.091,Z 394.659,A -85,B 0,C 180,E1 -11565.992,E2 -11565.992} C_VEL
LIN {X 0,Y 390.684,Z 398.584,A -85,B 0,C 180,E1 -11569.072,E2 -11569.072} C_VEL
LIN {X 0,Y 390.854,Z 401.17,A -85,B 0,C 180,E1 -11570.998,E2 -11570.998} C_VEL
LIN {X 0,Y 390.742,Z 404.835,A -85,B 0,C 180,E1 -11573.591,E2 -11573.591} C_VEL
LIN {X 0,Y 390.476,Z 408.498,A -85,B 0,C 180,E1 -11576.085,E2 -11576.085} C_VEL
LIN {X 0,Y 390.171,Z 412.163,A -85,B 0,C 180,E1 -11578.509,E2 -11578.509} C_VEL
LIN {X 0,Y 389.814,Z 417.695,A -85,B 0,C 180,E1 -11582.059,E2 -11582.059} C_VEL
LIN {X 0,Y 389.457,Z 423.19,A -85,B 0,C 180,E1 -11585.477,E2 -11585.477} C_VEL
LIN {X 0,Y 389.322,Z 426.451,A -85,B 0,C 180,E1 -11587.467,E2 -11587.467} C_VEL
LIN {X 0,Y 393.34,Z 441.755,A -85,B 0,C 180,E1 -11588.162,E2 -11588.162} C_VEL
LIN {X 0,Y 396.3,Z 456.005,A -85,B 0,C 180,E1 -11588.979,E2 -11588.979} C_VEL
LIN {X 0,Y 397.195,Z 462.428,A -85,B 0,C 180,E1 -11589.398,E2 -11589.398} C_VEL
LIN {X 0,Y 396.214,Z 476.073,A -85,B 0,C 180,E1 -11590.304,E2 -11590.304} C_VEL
LIN {X 0,Y 395.056,Z 488.193,A -85,B 0,C 180,E1 -11591.324,E2 -11591.324} C_VEL
LIN {X 0,Y 393.768,Z 500.423,A -85,B 0,C 180,E1 -11592.605,E2 -11592.605} C_VEL
LIN {X 0,Y 392.676,Z 510.517,A -85,B 0,C 180,E1 -11593.894,E2 -11593.894} C_VEL
LIN {X 0,Y 391.575,Z 520.552,A -85,B 0,C 180,E1 -11595.447,E2 -11595.447} C_VEL
LIN {X 0,Y 390.736,Z 528.887,A -85,B 0,C 180,E1 -11597.007,E2 -11597.007} C_VEL
LIN {X 0,Y 389.881,Z 536.853,A -85,B 0,C 180,E1 -11598.826,E2 -11598.826} C_VEL
LIN {X 0,Y 389.343,Z 543.269,A -85,B 0,C 180,E1 -11600.65,E2 -11600.65} C_VEL
LIN {X 0,Y 388.928,Z 548.955,A -85,B 0,C 180,E1 -11602.733,E2 -11602.733} C_VEL
LIN {X 0,Y 388.738,Z 553.081,A -85,B 0,C 180,E1 -11604.814,E2 -11604.814} C_VEL
LIN {X 0,Y 388.596,Z 555.774,A -85,B 0,C 180,E1 -11606.89,E2 -11606.89} C_VEL
LIN {X 0,Y 388.653,Z 557.109,A -85,B 0,C 180,E1 -11608.964,E2 -11608.964} C_VEL
LIN {X 0,Y 388.653,Z 557.108,A -85,B 0,C 180,E1 -11611.036,E2 -11611.036} C_VEL
LIN {X 0,Y 388.596,Z 555.771,A -85,B 0,C 180,E1 -11613.11,E2 -11613.11} C_VEL
LIN {X 0,Y 388.741,Z 553.075,A -85,B 0,C 180,E1 -11615.186,E2 -11615.186} C_VEL
LIN {X 0,Y 388.929,Z 548.941,A -85,B 0,C 180,E1 -11617.267,E2 -11617.267} C_VEL
LIN {X 0,Y 389.336,Z 543.247,A -85,B 0,C 180,E1 -11619.35,E2 -11619.35} C_VEL
LIN {X 0,Y 389.88,Z 536.829,A -85,B 0,C 180,E1 -11621.173,E2 -11621.173} C_VEL
LIN {X 0,Y 390.734,Z 528.855,A -85,B 0,C 180,E1 -11622.993,E2 -11622.993} C_VEL
LIN {X 0,Y 391.593,Z 520.513,A -85,B 0,C 180,E1 -11624.552,E2 -11624.552} C_VEL
LIN {X 0,Y 392.672,Z 510.47,A -85,B 0,C 180,E1 -11626.106,E2 -11626.106} C_VEL
LIN {X 0,Y 393.892,Z 499.265,A -85,B 0,C 180,E1 -11627.523,E2 -11627.523} C_VEL
LIN {X 0,Y 395.23,Z 486.692,A -85,B 0,C 180,E1 -11628.802,E2 -11628.802} C_VEL
LIN {X 0,Y 396.361,Z 473.917,A -85,B 0,C 180,E1 -11629.845,E2 -11629.845} C_VEL
LIN {X 0,Y 397.151,Z 462.169,A -85,B 0,C 180,E1 -11630.611,E2 -11630.611} C_VEL
LIN {X 0,Y 395.485,Z 451.902,A -85,B 0,C 180,E1 -11631.271,E2 -11631.271} C_VEL
LIN {X 0,Y 392.507,Z 438.376,A -85,B 0,C 180,E1 -11632.004,E2 -11632.004} C_VEL
LIN {X 0,Y 389.335,Z 426.396,A -85,B 0,C 180,E1 -11632.557,E2 -11632.557} C_VEL
LIN {X 0,Y 389.565,Z 421.331,A -85,B 0,C 180,E1 -11635.656,E2 -11635.656} C_VEL
LIN {X 0,Y 389.934,Z 415.813,A -85,B 0,C 180,E1 -11639.12,E2 -11639.12} C_VEL
LIN {X 0,Y 390.301,Z 410.317,A -85,B 0,C 180,E1 -11642.697,E2 -11642.697} C_VEL
LIN {X 0,Y 390.672,Z 405.479,A -85,B 0,C 180,E1 -11645.95,E2 -11645.95} C_VEL
LIN {X 0,Y 390.851,Z 402.945,A -85,B 0,C 180,E1 -11647.704,E2 -11647.704} C_VEL
LIN {X 0,Y 390.751,Z 399.319,A -85,B 0,C 180,E1 -11650.353,E2 -11650.353} C_VEL
LIN {X 0,Y 390.225,Z 395.662,A -85,B 0,C 180,E1 -11653.187,E2 -11653.187} C_VEL
LIN {X 0,Y 390.089,Z 394.523,A -85,B 0,C 180,E1 -11654.215,E2 -11654.215} C_VEL
LIN {X 0,Y 390.081,Z 394.525,A -85,B 0,C 180,E1 -11657.62,E2 -11657.62} C_VEL
LIN {X 0,Y 390.096,Z 394.521,A -85,B 0,C 180,E1 -11660.908,E2 -11660.908} C_VEL
LIN {X 0,Y 390.087,Z 394.521,A -85,B 0,C 180,E1 -11664.793,E2 -11664.793} C_VEL
LIN {X 0,Y 390.032,Z 394.528,A -85,B 0,C 180,E1 -11667.875,E2 -11667.875} C_VEL
LIN {X 0,Y 390.06,Z 394.526,A -85,B 0,C 180,E1 -11670.891,E2 -11670.891} C_VEL
LIN {X 0,Y 390.12,Z 394.517,A -85,B 0,C 180,E1 -11674.257,E2 -11674.257} C_VEL
LIN {X 0,Y 390.038,Z 394.525,A -85,B 0,C 180,E1 -11677.766,E2 -11677.766} C_VEL
LIN {X 0,Y 390.107,Z 394.516,A -85,B 0,C 180,E1 -11681.078,E2 -11681.078} C_VEL
LIN {X 0,Y 390.146,Z 394.511,A -85,B 0,C 180,E1 -11684.323,E2 -11684.323} C_VEL
LIN {X 0,Y 390.172,Z 394.508,A -85,B 0,C 180,E1 -11687.517,E2 -11687.517} C_VEL
LIN {X 0,Y 390.316,Z 394.493,A -85,B 0,C 180,E1 -11691.718,E2 -11691.718} C_VEL
LIN {X 0,Y 390.332,Z 394.49,A -85,B 0,C 180,E1 -11693.798,E2 -11693.798} C_VEL
LIN {X 0,Y 390.422,Z 394.477,A -85,B 0,C 180,E1 -11697.937,E2 -11697.937} C_VEL
LIN {X 0,Y 390.552,Z 394.463,A -85,B 0,C 180,E1 -11700,E2 -11700} C_VEL
LIN {X 0,Y 390.312,Z 394.493,A -85,B 0,C 180,E1 -11703.097,E2 -11703.097} C_VEL
LIN {X 0,Y 390.311,Z 394.489,A -85,B 0,C 180,E1 -11706.653,E2 -11706.653} C_VEL
LIN {X 0,Y 390.21,Z 394.504,A -85,B 0,C 180,E1 -11709.329,E2 -11709.329} C_VEL
LIN {X 0,Y 390.196,Z 394.502,A -85,B 0,C 180,E1 -11713.439,E2 -11713.439} C_VEL
LIN {X 0,Y 390.152,Z 394.507,A -85,B 0,C 180,E1 -11717.309,E2 -11717.309} C_VEL
LIN {X 0,Y 390.089,Z 394.518,A -85,B 0,C 180,E1 -11720.47,E2 -11720.47} C_VEL
LIN {X 0,Y 390.091,Z 394.518,A -85,B 0,C 180,E1 -11723.351,E2 -11723.351} C_VEL
LIN {X 0,Y 390.115,Z 394.515,A -85,B 0,C 180,E1 -11726.768,E2 -11726.768} C_VEL
LIN {X 0,Y 390.04,Z 394.524,A -85,B 0,C 180,E1 -11730.3,E2 -11730.3} C_VEL
LIN {X 0,Y 390.07,Z 394.524,A -85,B 0,C 180,E1 -11734.025,E2 -11734.025} C_VEL
LIN {X 0,Y 390.047,Z 394.525,A -85,B 0,C 180,E1 -11737.551,E2 -11737.551} C_VEL
LIN {X 0,Y 390.057,Z 394.524,A -85,B 0,C 180,E1 -11740.821,E2 -11740.821} C_VEL
LIN {X 0,Y 390.056,Z 394.523,A -85,B 0,C 180,E1 -11743.886,E2 -11743.886} C_VEL
LIN {X 0,Y 390.062,Z 394.524,A -85,B 0,C 180,E1 -11746.79,E2 -11746.79} C_VEL
LIN {X 0,Y 390.054,Z 394.67,A -85,B 0,C 180,E1 -11748.19,E2 -11748.19} C_VEL
LIN {X 0,Y 390.364,Z 397.881,A -85,B 0,C 180,E1 -11750.94,E2 -11750.94} C_VEL
LIN {X 0,Y 390.334,Z 401.083,A -85,B 0,C 180,E1 -11753.547,E2 -11753.547} C_VEL
LIN {X 0,Y 390.164,Z 404.283,A -85,B 0,C 180,E1 -11756.055,E2 -11756.055} C_VEL
LIN {X 0,Y 389.957,Z 407.472,A -85,B 0,C 180,E1 -11758.49,E2 -11758.49} C_VEL
LIN {X 0,Y 389.667,Z 412.348,A -85,B 0,C 180,E1 -11762.1,E2 -11762.1} C_VEL
LIN {X 0,Y 389.403,Z 417.039,A -85,B 0,C 180,E1 -11765.474,E2 -11765.474} C_VEL
LIN {X 0,Y 389.318,Z 419.953,A -85,B 0,C 180,E1 -11767.535,E2 -11767.535} C_VEL
LIN {X 0,Y 393.243,Z 434.012,A -85,B 0,C 180,E1 -11768.186,E2 -11768.186} C_VEL
LIN {X 0,Y 396.368,Z 447.962,A -85,B 0,C 180,E1 -11768.992,E2 -11768.992} C_VEL
LIN {X 0,Y 397.431,Z 453.833,A -85,B 0,C 180,E1 -11769.382,E2 -11769.382} C_VEL
LIN {X 0,Y 396.55,Z 467.054,A -85,B 0,C 180,E1 -11770.239,E2 -11770.239} C_VEL
LIN {X 0,Y 395.501,Z 478.954,A -85,B 0,C 180,E1 -11771.211,E2 -11771.211} C_VEL
LIN {X 0,Y 394.282,Z 490.411,A -85,B 0,C 180,E1 -11772.361,E2 -11772.361} C_VEL
LIN {X 0,Y 393.124,Z 500.925,A -85,B 0,C 180,E1 -11773.646,E2 -11773.646} C_VEL
LIN {X 0,Y 391.961,Z 511.364,A -85,B 0,C 180,E1 -11775.196,E2 -11775.196} C_VEL
LIN {X 0,Y 391.123,Z 519.973,A -85,B 0,C 180,E1 -11776.756,E2 -11776.756} C_VEL
LIN {X 0,Y 390.145,Z 528.227,A -85,B 0,C 180,E1 -11778.571,E2 -11778.571} C_VEL
LIN {X 0,Y 389.634,Z 533.976,A -85,B 0,C 180,E1 -11780.133,E2 -11780.133} C_VEL
LIN {X 0,Y 389.208,Z 538.705,A -85,B 0,C 180,E1 -11781.694,E2 -11781.694} C_VEL
LIN {X 0,Y 388.923,Z 543.602,A -85,B 0,C 180,E1 -11783.776,E2 -11783.776} C_VEL
LIN {X 0,Y 388.715,Z 547.012,A -85,B 0,C 180,E1 -11785.853,E2 -11785.853} C_VEL
LIN {X 0,Y 388.66,Z 549.037,A -85,B 0,C 180,E1 -11787.928,E2 -11787.928} C_VEL
LIN {X 0,Y 388.672,Z 549.732,A -85,B 0,C 180,E1 -11790,E2 -11790} C_VEL
LIN {X 0,Y 388.659,Z 549.106,A -85,B 0,C 180,E1 -11792.073,E2 -11792.073} C_VEL
LIN {X 0,Y 388.713,Z 547.142,A -85,B 0,C 180,E1 -11794.147,E2 -11794.147} C_VEL
LIN {X 0,Y 388.923,Z 543.795,A -85,B 0,C 180,E1 -11796.225,E2 -11796.225} C_VEL
LIN {X 0,Y 389.205,Z 538.968,A -85,B 0,C 180,E1 -11798.306,E2 -11798.306} C_VEL
LIN {X 0,Y 389.794,Z 532.505,A -85,B 0,C 180,E1 -11800.387,E2 -11800.387} C_VEL
LIN {X 0,Y 390.55,Z 525.307,A -85,B 0,C 180,E1 -11802.207,E2 -11802.207} C_VEL
LIN {X 0,Y 391.333,Z 517.834,A -85,B 0,C 180,E1 -11803.753,E2 -11803.753} C_VEL
LIN {X 0,Y 392.273,Z 508.709,A -85,B 0,C 180,E1 -11805.323,E2 -11805.323} C_VEL
LIN {X 0,Y 393.507,Z 497.737,A -85,B 0,C 180,E1 -11806.871,E2 -11806.871} C_VEL
LIN {X 0,Y 394.731,Z 486.548,A -85,B 0,C 180,E1 -11808.155,E2 -11808.155} C_VEL
LIN {X 0,Y 395.423,Z 479.988,A -85,B 0,C 180,E1 -11808.792,E2 -11808.792} C_VEL
LIN {X 0,Y 395.499,Z 475.035,A -85,B 0,C 180,E1 -11809.254,E2 -11809.254} C_VEL
LIN {X 0,Y 393.993,Z 466.814,A -85,B 0,C 180,E1 -11810.014,E2 -11810.014} C_VEL
LIN {X 0,Y 392.138,Z 460.182,A -85,B 0,C 180,E1 -11810.601,E2 -11810.601} C_VEL
LIN {X 0,Y 390.485,Z 453.307,A -85,B 0,C 180,E1 -11811.139,E2 -11811.139} C_VEL
LIN {X 0,Y 387.51,Z 439.204,A -85,B 0,C 180,E1 -11812.048,E2 -11812.048} C_VEL
LIN {X 0,Y 383.613,Z 424.867,A -85,B 0,C 180,E1 -11812.802,E2 -11812.802} C_VEL
LIN {X 0,Y 382.232,Z 420.003,A -85,B 0,C 180,E1 -11813.025,E2 -11813.025} C_VEL
LIN {X 0,Y 382.481,Z 415.652,A -85,B 0,C 180,E1 -11816.168,E2 -11816.168} C_VEL
LIN {X 0,Y 382.712,Z 410.86,A -85,B 0,C 180,E1 -11819.724,E2 -11819.724} C_VEL
LIN {X 0,Y 382.998,Z 407.319,A -85,B 0,C 180,E1 -11822.424,E2 -11822.424} C_VEL
LIN {X 0,Y 383.263,Z 402.881,A -85,B 0,C 180,E1 -11825.93,E2 -11825.93} C_VEL
LIN {X 0,Y 383.342,Z 399.662,A -85,B 0,C 180,E1 -11828.561,E2 -11828.561} C_VEL
LIN {X 0,Y 383.162,Z 396.446,A -85,B 0,C 180,E1 -11831.324,E2 -11831.324} C_VEL
LIN {X 0,Y 383.034,Z 395.401,A -85,B 0,C 180,E1 -11832.783,E2 -11832.783} C_VEL
LIN {X 0,Y 383,Z 395.405,A -85,B 0,C 180,E1 -11835.789,E2 -11835.789} C_VEL
LIN {X 0,Y 382.99,Z 395.406,A -85,B 0,C 180,E1 -11838.796,E2 -11838.796} C_VEL
LIN {X 0,Y 383.004,Z 395.401,A -85,B 0,C 180,E1 -11842.096,E2 -11842.096} C_VEL
LIN {X 0,Y 383.021,Z 395.399,A -85,B 0,C 180,E1 -11845.332,E2 -11845.332} C_VEL
LIN {X 0,Y 382.985,Z 395.405,A -85,B 0,C 180,E1 -11849.081,E2 -11849.081} C_VEL
LIN {X 0,Y 383.059,Z 395.396,A -85,B 0,C 180,E1 -11852.698,E2 -11852.698} C_VEL
LIN {X 0,Y 383.036,Z 395.395,A -85,B 0,C 180,E1 -11856.193,E2 -11856.193} C_VEL
LIN {X 0,Y 383.058,Z 395.39,A -85,B 0,C 180,E1 -11859.598,E2 -11859.598} C_VEL
LIN {X 0,Y 383.108,Z 395.388,A -85,B 0,C 180,E1 -11862.931,E2 -11862.931} C_VEL
LIN {X 0,Y 383.128,Z 395.385,A -85,B 0,C 180,E1 -11866.464,E2 -11866.464} C_VEL
LIN {X 0,Y 383.154,Z 395.383,A -85,B 0,C 180,E1 -11870.498,E2 -11870.498} C_VEL
LIN {X 0,Y 383.276,Z 395.367,A -85,B 0,C 180,E1 -11872.625,E2 -11872.625} C_VEL
LIN {X 0,Y 383.202,Z 395.377,A -85,B 0,C 180,E1 -11874.738,E2 -11874.738} C_VEL
LIN {X 0,Y 383.388,Z 395.353,A -85,B 0,C 180,E1 -11877.899,E2 -11877.899} C_VEL
LIN {X 0,Y 383.521,Z 395.34,A -85,B 0,C 180,E1 -11880,E2 -11880} C_VEL
LIN {X 0,Y 383.254,Z 395.372,A -85,B 0,C 180,E1 -11883.154,E2 -11883.154} C_VEL
LIN {X 0,Y 383.29,Z 395.366,A -85,B 0,C 180,E1 -11886.316,E2 -11886.316} C_VEL
LIN {X 0,Y 383.263,Z 395.37,A -85,B 0,C 180,E1 -11888.436,E2 -11888.436} C_VEL
LIN {X 0,Y 383.101,Z 395.39,A -85,B 0,C 180,E1 -11891.642,E2 -11891.642} C_VEL
LIN {X 0,Y 383.113,Z 395.389,A -85,B 0,C 180,E1 -11894.882,E2 -11894.882} C_VEL
LIN {X 0,Y 383.092,Z 395.391,A -85,B 0,C 180,E1 -11898.172,E2 -11898.172} C_VEL
LIN {X 0,Y 382.996,Z 395.403,A -85,B 0,C 180,E1 -11901.531,E2 -11901.531} C_VEL
LIN {X 0,Y 383.055,Z 395.394,A -85,B 0,C 180,E1 -11904.96,E2 -11904.96} C_VEL
LIN {X 0,Y 383.019,Z 395.399,A -85,B 0,C 180,E1 -11908.494,E2 -11908.494} C_VEL
LIN {X 0,Y 383.011,Z 395.402,A -85,B 0,C 180,E1 -11912.149,E2 -11912.149} C_VEL
LIN {X 0,Y 383.02,Z 395.401,A -85,B 0,C 180,E1 -11914.668,E2 -11914.668} C_VEL
LIN {X 0,Y 383.006,Z 395.405,A -85,B 0,C 180,E1 -11917.904,E2 -11917.904} C_VEL
LIN {X 0,Y 383.015,Z 395.403,A -85,B 0,C 180,E1 -11921.343,E2 -11921.343} C_VEL
LIN {X 0,Y 382.998,Z 395.405,A -85,B 0,C 180,E1 -11924.303,E2 -11924.303} C_VEL
LIN {X 0,Y 383.052,Z 395.508,A -85,B 0,C 180,E1 -11925.688,E2 -11925.688} C_VEL
LIN {X 0,Y 383.609,Z 399.295,A -85,B 0,C 180,E1 -11928.734,E2 -11928.734} C_VEL
LIN {X 0,Y 383.822,Z 402.953,A -85,B 0,C 180,E1 -11931.496,E2 -11931.496} C_VEL
LIN {X 0,Y 383.626,Z 406.604,A -85,B 0,C 180,E1 -11934.109,E2 -11934.109} C_VEL
LIN {X 0,Y 383.235,Z 412.112,A -85,B 0,C 180,E1 -11937.871,E2 -11937.871} C_VEL
LIN {X 0,Y 382.783,Z 418.082,A -85,B 0,C 180,E1 -11941.799,E2 -11941.799} C_VEL
LIN {X 0,Y 382.424,Z 423.125,A -85,B 0,C 180,E1 -11944.996,E2 -11944.996} C_VEL
LIN {X 0,Y 382.277,Z 426.377,A -85,B 0,C 180,E1 -11947.028,E2 -11947.028} C_VEL
LIN {X 0,Y 386.288,Z 441.409,A -85,B 0,C 180,E1 -11947.731,E2 -11947.731} C_VEL
LIN {X 0,Y 389.197,Z 454.938,A -85,B 0,C 180,E1 -11948.524,E2 -11948.524} C_VEL
LIN {X 0,Y 390.498,Z 463.664,A -85,B 0,C 180,E1 -11949.107,E2 -11949.107} C_VEL
LIN {X 0,Y 389.538,Z 476.009,A -85,B 0,C 180,E1 -11949.953,E2 -11949.953} C_VEL
LIN {X 0,Y 388.319,Z 488.128,A -85,B 0,C 180,E1 -11950.987,E2 -11950.987} C_VEL
LIN {X 0,Y 386.973,Z 500.356,A -85,B 0,C 180,E1 -11952.29,E2 -11952.29} C_VEL
LIN {X 0,Y 385.839,Z 510.45,A -85,B 0,C 180,E1 -11953.601,E2 -11953.601} C_VEL
LIN {X 0,Y 384.64,Z 520.484,A -85,B 0,C 180,E1 -11955.179,E2 -11955.179} C_VEL
LIN {X 0,Y 383.756,Z 528.819,A -85,B 0,C 180,E1 -11956.766,E2 -11956.766} C_VEL
LIN {X 0,Y 382.865,Z 536.785,A -85,B 0,C 180,E1 -11958.619,E2 -11958.619} C_VEL
LIN {X 0,Y 382.318,Z 543.201,A -85,B 0,C 180,E1 -11960.477,E2 -11960.477} C_VEL
LIN {X 0,Y 381.855,Z 548.886,A -85,B 0,C 180,E1 -11962.598,E2 -11962.598} C_VEL
LIN {X 0,Y 381.646,Z 553.012,A -85,B 0,C 180,E1 -11964.717,E2 -11964.717} C_VEL
LIN {X 0,Y 381.51,Z 555.706,A -85,B 0,C 180,E1 -11966.832,E2 -11966.832} C_VEL
LIN {X 0,Y 381.551,Z 557.041,A -85,B 0,C 180,E1 -11968.944,E2 -11968.944} C_VEL
LIN {X 0,Y 381.551,Z 557.039,A -85,B 0,C 180,E1 -11971.055,E2 -11971.055} C_VEL
LIN {X 0,Y 381.51,Z 555.702,A -85,B 0,C 180,E1 -11973.168,E2 -11973.168} C_VEL
LIN {X 0,Y 381.65,Z 553.005,A -85,B 0,C 180,E1 -11975.283,E2 -11975.283} C_VEL
LIN {X 0,Y 381.792,Z 550.056,A -85,B 0,C 180,E1 -11976.872,E2 -11976.872} C_VEL
LIN {X 0,Y 382.166,Z 544.79,A -85,B 0,C 180,E1 -11978.993,E2 -11978.993} C_VEL
LIN {X 0,Y 382.585,Z 539.694,A -85,B 0,C 180,E1 -11980.585,E2 -11980.585} C_VEL
LIN {X 0,Y 383.405,Z 532.424,A -85,B 0,C 180,E1 -11982.438,E2 -11982.438} C_VEL
LIN {X 0,Y 384.264,Z 523.796,A -85,B 0,C 180,E1 -11984.224,E2 -11984.224} C_VEL
LIN {X 0,Y 385.381,Z 513.966,A -85,B 0,C 180,E1 -11985.875,E2 -11985.875} C_VEL
LIN {X 0,Y 386.586,Z 503.503,A -85,B 0,C 180,E1 -11987.319,E2 -11987.319} C_VEL
LIN {X 0,Y 387.912,Z 491.956,A -85,B 0,C 180,E1 -11988.622,E2 -11988.622} C_VEL
LIN {X 0,Y 389.202,Z 479.144,A -85,B 0,C 180,E1 -11989.79,E2 -11989.79} C_VEL
LIN {X 0,Y 390.292,Z 466.144,A -85,B 0,C 180,E1 -11990.728,E2 -11990.728} C_VEL
LIN {X 0,Y 390.243,Z 461.195,A -85,B 0,C 180,E1 -11991.048,E2 -11991.048} C_VEL
LIN {X 0,Y 387.628,Z 447.278,A -85,B 0,C 180,E1 -11991.935,E2 -11991.935} C_VEL
LIN {X 0,Y 384.174,Z 433.308,A -85,B 0,C 180,E1 -11992.663,E2 -11992.663} C_VEL
LIN {X 0,Y 382.287,Z 426.357,A -85,B 0,C 180,E1 -11992.974,E2 -11992.974} C_VEL
LIN {X 0,Y 382.538,Z 421.268,A -85,B 0,C 180,E1 -11996.163,E2 -11996.163} C_VEL
LIN {X 0,Y 382.805,Z 417.581,A -85,B 0,C 180,E1 -11998.512,E2 -11998.512} C_VEL
LIN {X 0,Y 383.235,Z 412.091,A -85,B 0,C 180,E1 -12002.128,E2 -12002.128} C_VEL
LIN {X 0,Y 383.625,Z 406.58,A -85,B 0,C 180,E1 -12005.891,E2 -12005.891} C_VEL
LIN {X 0,Y 383.821,Z 402.928,A -85,B 0,C 180,E1 -12008.503,E2 -12008.503} C_VEL
LIN {X 0,Y 383.799,Z 401.103,A -85,B 0,C 180,E1 -12009.86,E2 -12009.86} C_VEL
LIN {X 0,Y 383.302,Z 397.306,A -85,B 0,C 180,E1 -12012.826,E2 -12012.826} C_VEL
LIN {X 0,Y 383.032,Z 395.402,A -85,B 0,C 180,E1 -12014.453,E2 -12014.453} C_VEL
LIN {X 0,Y 383.04,Z 395.401,A -85,B 0,C 180,E1 -12017.244,E2 -12017.244} C_VEL
LIN {X 0,Y 383.023,Z 395.4,A -85,B 0,C 180,E1 -12020.412,E2 -12020.412} C_VEL
LIN {X 0,Y 383.028,Z 395.401,A -85,B 0,C 180,E1 -12024.045,E2 -12024.045} C_VEL
LIN {X 0,Y 382.987,Z 395.408,A -85,B 0,C 180,E1 -12027.578,E2 -12027.578} C_VEL
LIN {X 0,Y 382.993,Z 395.404,A -85,B 0,C 180,E1 -12030.3,E2 -12030.3} C_VEL
LIN {X 0,Y 383.081,Z 395.395,A -85,B 0,C 180,E1 -12034.021,E2 -12034.021} C_VEL
LIN {X 0,Y 382.996,Z 395.405,A -85,B 0,C 180,E1 -12037.334,E2 -12037.334} C_VEL
LIN {X 0,Y 383.062,Z 395.396,A -85,B 0,C 180,E1 -12040.716,E2 -12040.716} C_VEL
LIN {X 0,Y 383.087,Z 395.392,A -85,B 0,C 180,E1 -12044.027,E2 -12044.027} C_VEL
LIN {X 0,Y 383.138,Z 395.386,A -85,B 0,C 180,E1 -12047.284,E2 -12047.284} C_VEL
LIN {X 0,Y 383.153,Z 395.385,A -85,B 0,C 180,E1 -12050.498,E2 -12050.498} C_VEL
LIN {X 0,Y 383.275,Z 395.363,A -85,B 0,C 180,E1 -12052.625,E2 -12052.625} C_VEL
LIN {X 0,Y 383.201,Z 395.377,A -85,B 0,C 180,E1 -12054.739,E2 -12054.739} C_VEL
LIN {X 0,Y 383.39,Z 395.353,A -85,B 0,C 180,E1 -12057.899,E2 -12057.899} C_VEL
LIN {X 0,Y 383.521,Z 395.339,A -85,B 0,C 180,E1 -12060,E2 -12060} C_VEL
LIN {X 0,Y 383.248,Z 395.373,A -85,B 0,C 180,E1 -12063.154,E2 -12063.154} C_VEL
LIN {X 0,Y 383.271,Z 395.368,A -85,B 0,C 180,E1 -12066.647,E2 -12066.647} C_VEL
LIN {X 0,Y 383.262,Z 395.37,A -85,B 0,C 180,E1 -12068.436,E2 -12068.436} C_VEL
LIN {X 0,Y 383.1,Z 395.39,A -85,B 0,C 180,E1 -12071.642,E2 -12071.642} C_VEL
LIN {X 0,Y 383.115,Z 395.389,A -85,B 0,C 180,E1 -12074.882,E2 -12074.882} C_VEL
LIN {X 0,Y 383.091,Z 395.392,A -85,B 0,C 180,E1 -12078.172,E2 -12078.172} C_VEL
LIN {X 0,Y 382.995,Z 395.403,A -85,B 0,C 180,E1 -12081.531,E2 -12081.531} C_VEL
LIN {X 0,Y 383.054,Z 395.395,A -85,B 0,C 180,E1 -12084.96,E2 -12084.96} C_VEL
LIN {X 0,Y 383.019,Z 395.399,A -85,B 0,C 180,E1 -12088.495,E2 -12088.495} C_VEL
LIN {X 0,Y 383.011,Z 395.402,A -85,B 0,C 180,E1 -12092.15,E2 -12092.15} C_VEL
LIN {X 0,Y 383.02,Z 395.399,A -85,B 0,C 180,E1 -12094.668,E2 -12094.668} C_VEL
LIN {X 0,Y 383.003,Z 395.4,A -85,B 0,C 180,E1 -12097.904,E2 -12097.904} C_VEL
LIN {X 0,Y 382.985,Z 395.403,A -85,B 0,C 180,E1 -12101.347,E2 -12101.347} C_VEL
LIN {X 0,Y 382.999,Z 395.402,A -85,B 0,C 180,E1 -12104.304,E2 -12104.304} C_VEL
LIN {X 0,Y 383.011,Z 395.402,A -85,B 0,C 180,E1 -12107.24,E2 -12107.24} C_VEL
LIN {X 0,Y 383.136,Z 396.434,A -85,B 0,C 180,E1 -12108.771,E2 -12108.771} C_VEL
LIN {X 0,Y 383.337,Z 399.529,A -85,B 0,C 180,E1 -12111.439,E2 -12111.439} C_VEL
LIN {X 0,Y 383.269,Z 402.748,A -85,B 0,C 180,E1 -12114.071,E2 -12114.071} C_VEL
LIN {X 0,Y 383.003,Z 407.182,A -85,B 0,C 180,E1 -12117.575,E2 -12117.575} C_VEL
LIN {X 0,Y 382.711,Z 410.723,A -85,B 0,C 180,E1 -12120.276,E2 -12120.276} C_VEL
LIN {X 0,Y 382.481,Z 415.514,A -85,B 0,C 180,E1 -12123.833,E2 -12123.833} C_VEL
LIN {X 0,Y 382.273,Z 420.006,A -85,B 0,C 180,E1 -12127.082,E2 -12127.082} C_VEL
LIN {X 0,Y 386.861,Z 436.433,A -85,B 0,C 180,E1 -12127.897,E2 -12127.897} C_VEL
LIN {X 0,Y 389.823,Z 449.993,A -85,B 0,C 180,E1 -12128.726,E2 -12128.726} C_VEL
LIN {X 0,Y 390.727,Z 455.721,A -85,B 0,C 180,E1 -12129.122,E2 -12129.122} C_VEL
LIN {X 0,Y 389.794,Z 468.221,A -85,B 0,C 180,E1 -12129.966,E2 -12129.966} C_VEL
LIN {X 0,Y 388.604,Z 480.452,A -85,B 0,C 180,E1 -12131.002,E2 -12131.002} C_VEL
LIN {X 0,Y 387.377,Z 491.656,A -85,B 0,C 180,E1 -12132.172,E2 -12132.172} C_VEL
LIN {X 0,Y 386.075,Z 502.919,A -85,B 0,C 180,E1 -12133.611,E2 -12133.611} C_VEL
LIN {X 0,Y 384.891,Z 512.978,A -85,B 0,C 180,E1 -12135.189,E2 -12135.189} C_VEL
LIN {X 0,Y 384.052,Z 521.328,A -85,B 0,C 180,E1 -12136.777,E2 -12136.777} C_VEL
LIN {X 0,Y 383.05,Z 529.306,A -85,B 0,C 180,E1 -12138.625,E2 -12138.625} C_VEL
LIN {X 0,Y 382.441,Z 535.725,A -85,B 0,C 180,E1 -12140.48,E2 -12140.48} C_VEL
LIN {X 0,Y 381.96,Z 541.418,A -85,B 0,C 180,E1 -12142.6,E2 -12142.6} C_VEL
LIN {X 0,Y 381.752,Z 545.555,A -85,B 0,C 180,E1 -12144.719,E2 -12144.719} C_VEL
LIN {X 0,Y 381.551,Z 548.263,A -85,B 0,C 180,E1 -12146.832,E2 -12146.832} C_VEL
LIN {X 0,Y 381.558,Z 549.619,A -85,B 0,C 180,E1 -12148.945,E2 -12148.945} C_VEL
LIN {X 0,Y 381.557,Z 549.653,A -85,B 0,C 180,E1 -12151.056,E2 -12151.056} C_VEL
LIN {X 0,Y 381.55,Z 548.362,A -85,B 0,C 180,E1 -12153.168,E2 -12153.168} C_VEL
LIN {X 0,Y 381.749,Z 545.714,A -85,B 0,C 180,E1 -12155.282,E2 -12155.282} C_VEL
LIN {X 0,Y 381.959,Z 541.644,A -85,B 0,C 180,E1 -12157.4,E2 -12157.4} C_VEL
LIN {X 0,Y 382.416,Z 536.02,A -85,B 0,C 180,E1 -12159.521,E2 -12159.521} C_VEL
LIN {X 0,Y 383.011,Z 529.671,A -85,B 0,C 180,E1 -12161.377,E2 -12161.377} C_VEL
LIN {X 0,Y 384.018,Z 521.774,A -85,B 0,C 180,E1 -12163.225,E2 -12163.225} C_VEL
LIN {X 0,Y 384.858,Z 513.515,A -85,B 0,C 180,E1 -12164.813,E2 -12164.813} C_VEL
LIN {X 0,Y 386.04,Z 503.562,A -85,B 0,C 180,E1 -12166.391,E2 -12166.391} C_VEL
LIN {X 0,Y 387.314,Z 492.482,A -85,B 0,C 180,E1 -12167.831,E2 -12167.831} C_VEL
LIN {X 0,Y 388.638,Z 480.491,A -85,B 0,C 180,E1 -12169.09,E2 -12169.09} C_VEL
LIN {X 0,Y 389.811,Z 467.891,A -85,B 0,C 180,E1 -12170.157,E2 -12170.157} C_VEL
LIN {X 0,Y 390.735,Z 455.898,A -85,B 0,C 180,E1 -12170.966,E2 -12170.966} C_VEL
LIN {X 0,Y 390.485,Z 453.307,A -85,B 0,C 180,E1 -12171.139,E2 -12171.139} C_VEL
LIN {X 0,Y 388.966,Z 448.247,A -85,B 0,C 180,E1 -12171.523,E2 -12171.523} C_VEL
LIN {X 0,Y 384.762,Z 440.447,A -85,B 0,C 180,E1 -12172.168,E2 -12172.168} C_VEL
LIN {X 0,Y 379.058,Z 431.1,A -85,B 0,C 180,E1 -12172.896,E2 -12172.896} C_VEL
LIN {X 0,Y 377.439,Z 427.738,A -85,B 0,C 180,E1 -12173.107,E2 -12173.107} C_VEL
LIN {X 0,Y 375.186,Z 420.085,A -85,B 0,C 180,E1 -12173.472,E2 -12173.472} C_VEL
LIN {X 0,Y 375.444,Z 415.722,A -85,B 0,C 180,E1 -12176.696,E2 -12176.696} C_VEL
LIN {X 0,Y 375.738,Z 410.923,A -85,B 0,C 180,E1 -12180.333,E2 -12180.333} C_VEL
LIN {X 0,Y 375.983,Z 407.719,A -85,B 0,C 180,E1 -12182.825,E2 -12182.825} C_VEL
LIN {X 0,Y 376.274,Z 403.085,A -85,B 0,C 180,E1 -12186.568,E2 -12186.568} C_VEL
LIN {X 0,Y 376.285,Z 399.701,A -85,B 0,C 180,E1 -12189.422,E2 -12189.422} C_VEL
LIN {X 0,Y 375.998,Z 396.486,A -85,B 0,C 180,E1 -12192.291,E2 -12192.291} C_VEL
LIN {X 0,Y 375.931,Z 396.285,A -85,B 0,C 180,E1 -12195.268,E2 -12195.268} C_VEL
LIN {X 0,Y 375.936,Z 396.285,A -85,B 0,C 180,E1 -12198.399,E2 -12198.399} C_VEL
LIN {X 0,Y 375.978,Z 396.276,A -85,B 0,C 180,E1 -12201.729,E2 -12201.729} C_VEL
LIN {X 0,Y 375.983,Z 396.276,A -85,B 0,C 180,E1 -12205.333,E2 -12205.333} C_VEL
LIN {X 0,Y 375.96,Z 396.277,A -85,B 0,C 180,E1 -12208.438,E2 -12208.438} C_VEL
LIN {X 0,Y 375.986,Z 396.277,A -85,B 0,C 180,E1 -12212.14,E2 -12212.14} C_VEL
LIN {X 0,Y 376.009,Z 396.273,A -85,B 0,C 180,E1 -12214.539,E2 -12214.539} C_VEL
LIN {X 0,Y 375.966,Z 396.277,A -85,B 0,C 180,E1 -12218.046,E2 -12218.046} C_VEL
LIN {X 0,Y 376.027,Z 396.27,A -85,B 0,C 180,E1 -12221.474,E2 -12221.474} C_VEL
LIN {X 0,Y 376.062,Z 396.265,A -85,B 0,C 180,E1 -12224.833,E2 -12224.833} C_VEL
LIN {X 0,Y 376.053,Z 396.267,A -85,B 0,C 180,E1 -12228.137,E2 -12228.137} C_VEL
LIN {X 0,Y 376.26,Z 396.243,A -85,B 0,C 180,E1 -12231.877,E2 -12231.877} C_VEL
LIN {X 0,Y 376.174,Z 396.252,A -85,B 0,C 180,E1 -12234.64,E2 -12234.64} C_VEL
LIN {X 0,Y 376.355,Z 396.229,A -85,B 0,C 180,E1 -12237.86,E2 -12237.86} C_VEL
LIN {X 0,Y 376.49,Z 396.215,A -85,B 0,C 180,E1 -12240,E2 -12240} C_VEL
LIN {X 0,Y 376.192,Z 396.251,A -85,B 0,C 180,E1 -12243.213,E2 -12243.213} C_VEL
LIN {X 0,Y 376.25,Z 396.244,A -85,B 0,C 180,E1 -12246.435,E2 -12246.435} C_VEL
LIN {X 0,Y 376.209,Z 396.248,A -85,B 0,C 180,E1 -12248.595,E2 -12248.595} C_VEL
LIN {X 0,Y 376.053,Z 396.267,A -85,B 0,C 180,E1 -12251.863,E2 -12251.863} C_VEL
LIN {X 0,Y 376.061,Z 396.266,A -85,B 0,C 180,E1 -12255.167,E2 -12255.167} C_VEL
LIN {X 0,Y 376.026,Z 396.27,A -85,B 0,C 180,E1 -12258.526,E2 -12258.526} C_VEL
LIN {X 0,Y 375.966,Z 396.278,A -85,B 0,C 180,E1 -12261.954,E2 -12261.954} C_VEL
LIN {X 0,Y 376.009,Z 396.272,A -85,B 0,C 180,E1 -12265.461,E2 -12265.461} C_VEL
LIN {X 0,Y 375.963,Z 396.281,A -85,B 0,C 180,E1 -12269.08,E2 -12269.08} C_VEL
LIN {X 0,Y 375.953,Z 396.282,A -85,B 0,C 180,E1 -12272.828,E2 -12272.828} C_VEL
LIN {X 0,Y 375.961,Z 396.282,A -85,B 0,C 180,E1 -12275.415,E2 -12275.415} C_VEL
LIN {X 0,Y 375.98,Z 396.28,A -85,B 0,C 180,E1 -12278.271,E2 -12278.271} C_VEL
LIN {X 0,Y 375.962,Z 396.282,A -85,B 0,C 180,E1 -12281.605,E2 -12281.605} C_VEL
LIN {X 0,Y 376.035,Z 396.441,A -85,B 0,C 180,E1 -12285.443,E2 -12285.443} C_VEL
LIN {X 0,Y 376.668,Z 401.076,A -85,B 0,C 180,E1 -12289.228,E2 -12289.228} C_VEL
LIN {X 0,Y 376.791,Z 404.737,A -85,B 0,C 180,E1 -12292.01,E2 -12292.01} C_VEL
LIN {X 0,Y 376.482,Z 409.192,A -85,B 0,C 180,E1 -12295.222,E2 -12295.222} C_VEL
LIN {X 0,Y 376.094,Z 413.877,A -85,B 0,C 180,E1 -12298.451,E2 -12298.451} C_VEL
LIN {X 0,Y 375.686,Z 419.388,A -85,B 0,C 180,E1 -12302.116,E2 -12302.116} C_VEL
LIN {X 0,Y 375.306,Z 424.892,A -85,B 0,C 180,E1 -12305.671,E2 -12305.671} C_VEL
LIN {X 0,Y 375.287,Z 426.486,A -85,B 0,C 180,E1 -12306.581,E2 -12306.581} C_VEL
LIN {X 0,Y 379.19,Z 440.834,A -85,B 0,C 180,E1 -12307.271,E2 -12307.271} C_VEL
LIN {X 0,Y 382.045,Z 453.908,A -85,B 0,C 180,E1 -12308.049,E2 -12308.049} C_VEL
LIN {X 0,Y 383.775,Z 464.966,A -85,B 0,C 180,E1 -12308.815,E2 -12308.815} C_VEL
LIN {X 0,Y 382.698,Z 477.592,A -85,B 0,C 180,E1 -12309.719,E2 -12309.719} C_VEL
LIN {X 0,Y 381.277,Z 490.675,A -85,B 0,C 180,E1 -12310.902,E2 -12310.902} C_VEL
LIN {X 0,Y 379.935,Z 502.431,A -85,B 0,C 180,E1 -12312.229,E2 -12312.229} C_VEL
LIN {X 0,Y 378.755,Z 512.167,A -85,B 0,C 180,E1 -12313.562,E2 -12313.562} C_VEL
LIN {X 0,Y 377.592,Z 521.761,A -85,B 0,C 180,E1 -12315.145,E2 -12315.145} C_VEL
LIN {X 0,Y 376.702,Z 529.985,A -85,B 0,C 180,E1 -12316.788,E2 -12316.788} C_VEL
LIN {X 0,Y 375.775,Z 537.727,A -85,B 0,C 180,E1 -12318.675,E2 -12318.675} C_VEL
LIN {X 0,Y 375.263,Z 543.132,A -85,B 0,C 180,E1 -12320.296,E2 -12320.296} C_VEL
LIN {X 0,Y 374.788,Z 548.818,A -85,B 0,C 180,E1 -12322.457,E2 -12322.457} C_VEL
LIN {X 0,Y 374.558,Z 552.944,A -85,B 0,C 180,E1 -12324.617,E2 -12324.617} C_VEL
LIN {X 0,Y 374.427,Z 555.637,A -85,B 0,C 180,E1 -12326.772,E2 -12326.772} C_VEL
LIN {X 0,Y 374.45,Z 556.972,A -85,B 0,C 180,E1 -12328.924,E2 -12328.924} C_VEL
LIN {X 0,Y 374.45,Z 556.97,A -85,B 0,C 180,E1 -12331.075,E2 -12331.075} C_VEL
LIN {X 0,Y 374.427,Z 555.632,A -85,B 0,C 180,E1 -12333.228,E2 -12333.228} C_VEL
LIN {X 0,Y 374.565,Z 552.936,A -85,B 0,C 180,E1 -12335.383,E2 -12335.383} C_VEL
LIN {X 0,Y 374.728,Z 549.986,A -85,B 0,C 180,E1 -12337.002,E2 -12337.002} C_VEL
LIN {X 0,Y 375.119,Z 544.719,A -85,B 0,C 180,E1 -12339.163,E2 -12339.163} C_VEL
LIN {X 0,Y 375.555,Z 539.623,A -85,B 0,C 180,E1 -12340.786,E2 -12340.786} C_VEL
LIN {X 0,Y 376.442,Z 532.353,A -85,B 0,C 180,E1 -12342.672,E2 -12342.672} C_VEL
LIN {X 0,Y 377.388,Z 523.275,A -85,B 0,C 180,E1 -12344.574,E2 -12344.574} C_VEL
LIN {X 0,Y 378.509,Z 513.894,A -85,B 0,C 180,E1 -12346.171,E2 -12346.171} C_VEL
LIN {X 0,Y 379.806,Z 503.431,A -85,B 0,C 180,E1 -12347.638,E2 -12347.638} C_VEL
LIN {X 0,Y 381.146,Z 491.883,A -85,B 0,C 180,E1 -12348.965,E2 -12348.965} C_VEL
LIN {X 0,Y 382.52,Z 479.071,A -85,B 0,C 180,E1 -12350.151,E2 -12350.151} C_VEL
LIN {X 0,Y 383.608,Z 466.525,A -85,B 0,C 180,E1 -12351.074,E2 -12351.074} C_VEL
LIN {X 0,Y 383.517,Z 462.332,A -85,B 0,C 180,E1 -12351.36,E2 -12351.36} C_VEL
LIN {X 0,Y 380.848,Z 447.953,A -85,B 0,C 180,E1 -12352.311,E2 -12352.311} C_VEL
LIN {X 0,Y 377.389,Z 434.079,A -85,B 0,C 180,E1 -12353.066,E2 -12353.066} C_VEL
LIN {X 0,Y 375.262,Z 426.278,A -85,B 0,C 180,E1 -12353.436,E2 -12353.436} C_VEL
LIN {X 0,Y 375.514,Z 421.191,A -85,B 0,C 180,E1 -12356.691,E2 -12356.691} C_VEL
LIN {X 0,Y 375.788,Z 417.541,A -85,B 0,C 180,E1 -12359.095,E2 -12359.095} C_VEL
LIN {X 0,Y 376.093,Z 413.855,A -85,B 0,C 180,E1 -12361.549,E2 -12361.549} C_VEL
LIN {X 0,Y 376.536,Z 408.354,A -85,B 0,C 180,E1 -12365.353,E2 -12365.353} C_VEL
LIN {X 0,Y 376.809,Z 404.117,A -85,B 0,C 180,E1 -12368.431,E2 -12368.431} C_VEL
LIN {X 0,Y 376.661,Z 401.047,A -85,B 0,C 180,E1 -12370.772,E2 -12370.772} C_VEL
LIN {X 0,Y 376.033,Z 396.41,A -85,B 0,C 180,E1 -12374.557,E2 -12374.557} C_VEL
LIN {X 0,Y 375.961,Z 396.282,A -85,B 0,C 180,E1 -12378.395,E2 -12378.395} C_VEL
LIN {X 0,Y 375.979,Z 396.277,A -85,B 0,C 180,E1 -12381.729,E2 -12381.729} C_VEL
LIN {X 0,Y 375.981,Z 396.277,A -85,B 0,C 180,E1 -12385.333,E2 -12385.333} C_VEL
LIN {X 0,Y 375.958,Z 396.28,A -85,B 0,C 180,E1 -12388.438,E2 -12388.438} C_VEL
LIN {X 0,Y 375.984,Z 396.277,A -85,B 0,C 180,E1 -12392.14,E2 -12392.14} C_VEL
LIN {X 0,Y 376.006,Z 396.274,A -85,B 0,C 180,E1 -12394.539,E2 -12394.539} C_VEL
LIN {X 0,Y 375.959,Z 396.278,A -85,B 0,C 180,E1 -12398.046,E2 -12398.046} C_VEL
LIN {X 0,Y 376.025,Z 396.27,A -85,B 0,C 180,E1 -12401.474,E2 -12401.474} C_VEL
LIN {X 0,Y 376.063,Z 396.265,A -85,B 0,C 180,E1 -12404.833,E2 -12404.833} C_VEL
LIN {X 0,Y 376.052,Z 396.267,A -85,B 0,C 180,E1 -12408.137,E2 -12408.137} C_VEL
LIN {X 0,Y 376.259,Z 396.241,A -85,B 0,C 180,E1 -12411.877,E2 -12411.877} C_VEL
LIN {X 0,Y 376.173,Z 396.252,A -85,B 0,C 180,E1 -12414.64,E2 -12414.64} C_VEL
LIN {X 0,Y 376.356,Z 396.229,A -85,B 0,C 180,E1 -12417.86,E2 -12417.86} C_VEL
LIN {X 0,Y 376.491,Z 396.214,A -85,B 0,C 180,E1 -12420,E2 -12420} C_VEL
LIN {X 0,Y 376.187,Z 396.253,A -85,B 0,C 180,E1 -12423.213,E2 -12423.213} C_VEL
LIN {X 0,Y 376.235,Z 396.245,A -85,B 0,C 180,E1 -12426.638,E2 -12426.638} C_VEL
LIN {X 0,Y 376.207,Z 396.248,A -85,B 0,C 180,E1 -12428.595,E2 -12428.595} C_VEL
LIN {X 0,Y 376.052,Z 396.267,A -85,B 0,C 180,E1 -12431.863,E2 -12431.863} C_VEL
LIN {X 0,Y 376.063,Z 396.266,A -85,B 0,C 180,E1 -12435.167,E2 -12435.167} C_VEL
LIN {X 0,Y 376.026,Z 396.27,A -85,B 0,C 180,E1 -12438.526,E2 -12438.526} C_VEL
LIN {X 0,Y 375.965,Z 396.277,A -85,B 0,C 180,E1 -12441.954,E2 -12441.954} C_VEL
LIN {X 0,Y 376.008,Z 396.273,A -85,B 0,C 180,E1 -12445.461,E2 -12445.461} C_VEL
LIN {X 0,Y 375.962,Z 396.28,A -85,B 0,C 180,E1 -12449.08,E2 -12449.08} C_VEL
LIN {X 0,Y 375.952,Z 396.281,A -85,B 0,C 180,E1 -12452.828,E2 -12452.828} C_VEL
LIN {X 0,Y 375.96,Z 396.28,A -85,B 0,C 180,E1 -12455.415,E2 -12455.415} C_VEL
LIN {X 0,Y 375.977,Z 396.275,A -85,B 0,C 180,E1 -12458.271,E2 -12458.271} C_VEL
LIN {X 0,Y 375.935,Z 396.282,A -85,B 0,C 180,E1 -12461.601,E2 -12461.601} C_VEL
LIN {X 0,Y 375.956,Z 396.281,A -85,B 0,C 180,E1 -12465.264,E2 -12465.264} C_VEL
LIN {X 0,Y 375.968,Z 396.362,A -85,B 0,C 180,E1 -12467.705,E2 -12467.705} C_VEL
LIN {X 0,Y 376.275,Z 399.585,A -85,B 0,C 180,E1 -12470.577,E2 -12470.577} C_VEL
LIN {X 0,Y 376.276,Z 402.952,A -85,B 0,C 180,E1 -12473.432,E2 -12473.432} C_VEL
LIN {X 0,Y 376.088,Z 405.999,A -85,B 0,C 180,E1 -12475.902,E2 -12475.902} C_VEL
LIN {X 0,Y 375.777,Z 410.382,A -85,B 0,C 180,E1 -12479.353,E2 -12479.353} C_VEL
LIN {X 0,Y 375.557,Z 413.975,A -85,B 0,C 180,E1 -12482.106,E2 -12482.106} C_VEL
LIN {X 0,Y 375.249,Z 418.772,A -85,B 0,C 180,E1 -12485.667,E2 -12485.667} C_VEL
LIN {X 0,Y 375.209,Z 420.093,A -85,B 0,C 180,E1 -12486.638,E2 -12486.638} C_VEL
LIN {X 0,Y 379.278,Z 434.064,A -85,B 0,C 180,E1 -12487.334,E2 -12487.334} C_VEL
LIN {X 0,Y 382.366,Z 447.302,A -85,B 0,C 180,E1 -12488.139,E2 -12488.139} C_VEL
LIN {X 0,Y 384,Z 456.052,A -85,B 0,C 180,E1 -12488.754,E2 -12488.754} C_VEL
LIN {X 0,Y 383.126,Z 468.297,A -85,B 0,C 180,E1 -12489.602,E2 -12489.602} C_VEL
LIN {X 0,Y 381.886,Z 480.526,A -85,B 0,C 180,E1 -12490.655,E2 -12490.655} C_VEL
LIN {X 0,Y 380.616,Z 491.729,A -85,B 0,C 180,E1 -12491.845,E2 -12491.845} C_VEL
LIN {X 0,Y 379.248,Z 502.992,A -85,B 0,C 180,E1 -12493.307,E2 -12493.307} C_VEL
LIN {X 0,Y 378.004,Z 513.05,A -85,B 0,C 180,E1 -12494.913,E2 -12494.913} C_VEL
LIN {X 0,Y 377.109,Z 521.4,A -85,B 0,C 180,E1 -12496.529,E2 -12496.529} C_VEL
LIN {X 0,Y 376.065,Z 529.377,A -85,B 0,C 180,E1 -12498.411,E2 -12498.411} C_VEL
LIN {X 0,Y 375.42,Z 535.796,A -85,B 0,C 180,E1 -12500.3,E2 -12500.3} C_VEL
LIN {X 0,Y 374.89,Z 541.488,A -85,B 0,C 180,E1 -12502.46,E2 -12502.46} C_VEL
LIN {X 0,Y 374.661,Z 545.625,A -85,B 0,C 180,E1 -12504.618,E2 -12504.618} C_VEL
LIN {X 0,Y 374.467,Z 548.332,A -85,B 0,C 180,E1 -12506.772,E2 -12506.772} C_VEL
LIN {X 0,Y 374.457,Z 549.688,A -85,B 0,C 180,E1 -12508.925,E2 -12508.925} C_VEL
LIN {X 0,Y 374.457,Z 549.722,A -85,B 0,C 180,E1 -12511.076,E2 -12511.076} C_VEL
LIN {X 0,Y 374.466,Z 548.43,A -85,B 0,C 180,E1 -12513.228,E2 -12513.228} C_VEL
LIN {X 0,Y 374.658,Z 545.782,A -85,B 0,C 180,E1 -12515.382,E2 -12515.382} C_VEL
LIN {X 0,Y 374.816,Z 542.871,A -85,B 0,C 180,E1 -12517.001,E2 -12517.001} C_VEL
LIN {X 0,Y 375.238,Z 537.682,A -85,B 0,C 180,E1 -12519.161,E2 -12519.161} C_VEL
LIN {X 0,Y 375.76,Z 532.64,A -85,B 0,C 180,E1 -12520.78,E2 -12520.78} C_VEL
LIN {X 0,Y 376.62,Z 525.442,A -85,B 0,C 180,E1 -12522.666,E2 -12522.666} C_VEL
LIN {X 0,Y 377.488,Z 517.661,A -85,B 0,C 180,E1 -12524.33,E2 -12524.33} C_VEL
LIN {X 0,Y 378.526,Z 508.842,A -85,B 0,C 180,E1 -12525.894,E2 -12525.894} C_VEL
LIN {X 0,Y 379.922,Z 497.868,A -85,B 0,C 180,E1 -12527.494,E2 -12527.494} C_VEL
LIN {X 0,Y 381.223,Z 486.677,A -85,B 0,C 180,E1 -12528.822,E2 -12528.822} C_VEL
LIN {X 0,Y 382.562,Z 474.292,A -85,B 0,C 180,E1 -12530.009,E2 -12530.009} C_VEL
LIN {X 0,Y 383.659,Z 461.746,A -85,B 0,C 180,E1 -12530.973,E2 -12530.973} C_VEL
LIN {X 0,Y 384.012,Z 456.118,A -85,B 0,C 180,E1 -12531.341,E2 -12531.341} C_VEL
LIN {X 0,Y 381.403,Z 442.695,A -85,B 0,C 180,E1 -12532.259,E2 -12532.259} C_VEL
LIN {X 0,Y 377.686,Z 428.511,A -85,B 0,C 180,E1 -12533.067,E2 -12533.067} C_VEL
LIN {X 0,Y 377.439,Z 427.738,A -85,B 0,C 180,E1 -12533.107,E2 -12533.107} C_VEL
LIN {X 0,Y 375.938,Z 424.737,A -85,B 0,C 180,E1 -12533.383,E2 -12533.383} C_VEL
LIN {X 0,Y 373.967,Z 421.857,A -85,B 0,C 180,E1 -12533.89,E2 -12533.89} C_VEL
LIN {X 0,Y 372.113,Z 419.797,A -85,B 0,C 180,E1 -12534.511,E2 -12534.511} C_VEL
LIN {X 0,Y 370.216,Z 418.14,A -85,B 0,C 180,E1 -12535.372,E2 -12535.372} C_VEL
LIN {X 0,Y 368.626,Z 416.574,A -85,B 0,C 180,E1 -12536.615,E2 -12536.615} C_VEL
LIN {X 0,Y 368.416,Z 415.772,A -85,B 0,C 180,E1 -12537.25,E2 -12537.25} C_VEL
LIN {X 0,Y 368.773,Z 410.978,A -85,B 0,C 180,E1 -12540.968,E2 -12540.968} C_VEL
LIN {X 0,Y 368.991,Z 407.794,A -85,B 0,C 180,E1 -12543.529,E2 -12543.529} C_VEL
LIN {X 0,Y 369.268,Z 403.651,A -85,B 0,C 180,E1 -12546.931,E2 -12546.931} C_VEL
LIN {X 0,Y 369.218,Z 399.739,A -85,B 0,C 180,E1 -12550.33,E2 -12550.33} C_VEL
LIN {X 0,Y 369.027,Z 397.88,A -85,B 0,C 180,E1 -12552.034,E2 -12552.034} C_VEL
LIN {X 0,Y 368.898,Z 397.162,A -85,B 0,C 180,E1 -12553.618,E2 -12553.618} C_VEL
LIN {X 0,Y 368.888,Z 397.165,A -85,B 0,C 180,E1 -12556.696,E2 -12556.696} C_VEL
LIN {X 0,Y 368.914,Z 397.16,A -85,B 0,C 180,E1 -12559.643,E2 -12559.643} C_VEL
LIN {X 0,Y 368.905,Z 397.158,A -85,B 0,C 180,E1 -12563.144,E2 -12563.144} C_VEL
LIN {X 0,Y 368.901,Z 397.159,A -85,B 0,C 180,E1 -12566.462,E2 -12566.462} C_VEL
LIN {X 0,Y 368.931,Z 397.156,A -85,B 0,C 180,E1 -12569.047,E2 -12569.047} C_VEL
LIN {X 0,Y 368.978,Z 397.148,A -85,B 0,C 180,E1 -12571.564,E2 -12571.564} C_VEL
LIN {X 0,Y 369.003,Z 397.148,A -85,B 0,C 180,E1 -12574.02,E2 -12574.02} C_VEL
LIN {X 0,Y 368.935,Z 397.155,A -85,B 0,C 180,E1 -12577.605,E2 -12577.605} C_VEL
LIN {X 0,Y 368.985,Z 397.148,A -85,B 0,C 180,E1 -12581.107,E2 -12581.107} C_VEL
LIN {X 0,Y 369.001,Z 397.144,A -85,B 0,C 180,E1 -12584.535,E2 -12584.535} C_VEL
LIN {X 0,Y 369.008,Z 397.144,A -85,B 0,C 180,E1 -12587.907,E2 -12587.907} C_VEL
LIN {X 0,Y 369.232,Z 397.118,A -85,B 0,C 180,E1 -12591.8,E2 -12591.8} C_VEL
LIN {X 0,Y 369.147,Z 397.127,A -85,B 0,C 180,E1 -12594.538,E2 -12594.538} C_VEL
LIN {X 0,Y 369.319,Z 397.105,A -85,B 0,C 180,E1 -12597.819,E2 -12597.819} C_VEL
LIN {X 0,Y 369.46,Z 397.091,A -85,B 0,C 180,E1 -12600,E2 -12600} C_VEL
LIN {X 0,Y 369.322,Z 397.105,A -85,B 0,C 180,E1 -12602.181,E2 -12602.181} C_VEL
LIN {X 0,Y 369.211,Z 397.122,A -85,B 0,C 180,E1 -12606.558,E2 -12606.558} C_VEL
LIN {X 0,Y 369.141,Z 397.128,A -85,B 0,C 180,E1 -12608.761,E2 -12608.761} C_VEL
LIN {X 0,Y 369.008,Z 397.144,A -85,B 0,C 180,E1 -12612.093,E2 -12612.093} C_VEL
LIN {X 0,Y 369.001,Z 397.145,A -85,B 0,C 180,E1 -12615.465,E2 -12615.465} C_VEL
LIN {X 0,Y 368.985,Z 397.147,A -85,B 0,C 180,E1 -12618.893,E2 -12618.893} C_VEL
LIN {X 0,Y 368.935,Z 397.155,A -85,B 0,C 180,E1 -12622.395,E2 -12622.395} C_VEL
LIN {X 0,Y 369.002,Z 397.147,A -85,B 0,C 180,E1 -12625.98,E2 -12625.98} C_VEL
LIN {X 0,Y 368.917,Z 397.153,A -85,B 0,C 180,E1 -12629.69,E2 -12629.69} C_VEL
LIN {X 0,Y 368.9,Z 397.159,A -85,B 0,C 180,E1 -12633.043,E2 -12633.043} C_VEL
LIN {X 0,Y 368.921,Z 397.159,A -85,B 0,C 180,E1 -12636.196,E2 -12636.196} C_VEL
LIN {X 0,Y 368.911,Z 397.162,A -85,B 0,C 180,E1 -12638.952,E2 -12638.952} C_VEL
LIN {X 0,Y 368.911,Z 397.161,A -85,B 0,C 180,E1 -12642.014,E2 -12642.014} C_VEL
LIN {X 0,Y 368.983,Z 397.269,A -85,B 0,C 180,E1 -12645.096,E2 -12645.096} C_VEL
LIN {X 0,Y 369.523,Z 401.018,A -85,B 0,C 180,E1 -12648.266,E2 -12648.266} C_VEL
LIN {X 0,Y 369.784,Z 404.719,A -85,B 0,C 180,E1 -12651.19,E2 -12651.19} C_VEL
LIN {X 0,Y 369.604,Z 408.341,A -85,B 0,C 180,E1 -12653.881,E2 -12653.881} C_VEL
LIN {X 0,Y 369.125,Z 413.824,A -85,B 0,C 180,E1 -12657.784,E2 -12657.784} C_VEL
LIN {X 0,Y 368.728,Z 419.325,A -85,B 0,C 180,E1 -12661.543,E2 -12661.543} C_VEL
LIN {X 0,Y 368.262,Z 424.819,A -85,B 0,C 180,E1 -12665.174,E2 -12665.174} C_VEL
LIN {X 0,Y 368.224,Z 426.332,A -85,B 0,C 180,E1 -12666.102,E2 -12666.102} C_VEL
LIN {X 0,Y 372.192,Z 440.598,A -85,B 0,C 180,E1 -12666.812,E2 -12666.812} C_VEL
LIN {X 0,Y 375.008,Z 453.176,A -85,B 0,C 180,E1 -12667.577,E2 -12667.577} C_VEL
LIN {X 0,Y 377.004,Z 465.038,A -85,B 0,C 180,E1 -12668.426,E2 -12668.426} C_VEL
LIN {X 0,Y 376.183,Z 475.88,A -85,B 0,C 180,E1 -12669.209,E2 -12669.209} C_VEL
LIN {X 0,Y 374.883,Z 487.997,A -85,B 0,C 180,E1 -12670.278,E2 -12670.278} C_VEL
LIN {X 0,Y 373.397,Z 500.224,A -85,B 0,C 180,E1 -12671.623,E2 -12671.623} C_VEL
LIN {X 0,Y 372.18,Z 510.317,A -85,B 0,C 180,E1 -12672.981,E2 -12672.981} C_VEL
LIN {X 0,Y 370.854,Z 520.35,A -85,B 0,C 180,E1 -12674.614,E2 -12674.614} C_VEL
LIN {X 0,Y 369.826,Z 528.683,A -85,B 0,C 180,E1 -12676.258,E2 -12676.258} C_VEL
LIN {X 0,Y 369.058,Z 535.64,A -85,B 0,C 180,E1 -12677.908,E2 -12677.908} C_VEL
LIN {X 0,Y 368.388,Z 541.396,A -85,B 0,C 180,E1 -12679.558,E2 -12679.558} C_VEL
LIN {X 0,Y 367.953,Z 546.112,A -85,B 0,C 180,E1 -12681.211,E2 -12681.211} C_VEL
LIN {X 0,Y 367.563,Z 550.998,A -85,B 0,C 180,E1 -12683.412,E2 -12683.412} C_VEL
LIN {X 0,Y 367.424,Z 554.395,A -85,B 0,C 180,E1 -12685.612,E2 -12685.612} C_VEL
LIN {X 0,Y 367.314,Z 556.404,A -85,B 0,C 180,E1 -12687.807,E2 -12687.807} C_VEL
LIN {X 0,Y 367.372,Z 557.068,A -85,B 0,C 180,E1 -12690,E2 -12690} C_VEL
LIN {X 0,Y 367.314,Z 556.399,A -85,B 0,C 180,E1 -12692.193,E2 -12692.193} C_VEL
LIN {X 0,Y 367.426,Z 554.388,A -85,B 0,C 180,E1 -12694.388,E2 -12694.388} C_VEL
LIN {X 0,Y 367.587,Z 550.985,A -85,B 0,C 180,E1 -12696.587,E2 -12696.587} C_VEL
LIN {X 0,Y 367.949,Z 546.088,A -85,B 0,C 180,E1 -12698.789,E2 -12698.789} C_VEL
LIN {X 0,Y 368.533,Z 539.553,A -85,B 0,C 180,E1 -12700.994,E2 -12700.994} C_VEL
LIN {X 0,Y 369.483,Z 532.282,A -85,B 0,C 180,E1 -12702.915,E2 -12702.915} C_VEL
LIN {X 0,Y 370.433,Z 523.552,A -85,B 0,C 180,E1 -12704.787,E2 -12704.787} C_VEL
LIN {X 0,Y 371.674,Z 513.823,A -85,B 0,C 180,E1 -12706.477,E2 -12706.477} C_VEL
LIN {X 0,Y 373.032,Z 503.359,A -85,B 0,C 180,E1 -12707.969,E2 -12707.969} C_VEL
LIN {X 0,Y 374.414,Z 491.811,A -85,B 0,C 180,E1 -12709.319,E2 -12709.319} C_VEL
LIN {X 0,Y 375.843,Z 478.997,A -85,B 0,C 180,E1 -12710.525,E2 -12710.525} C_VEL
LIN {X 0,Y 376.97,Z 466.482,A -85,B 0,C 180,E1 -12711.461,E2 -12711.461} C_VEL
LIN {X 0,Y 376.399,Z 461.13,A -85,B 0,C 180,E1 -12711.855,E2 -12711.855} C_VEL
LIN {X 0,Y 373.776,Z 447.396,A -85,B 0,C 180,E1 -12712.779,E2 -12712.779} C_VEL
LIN {X 0,Y 370.303,Z 433.702,A -85,B 0,C 180,E1 -12713.544,E2 -12713.544} C_VEL
LIN {X 0,Y 368.229,Z 426.227,A -85,B 0,C 180,E1 -12713.896,E2 -12713.896} C_VEL
LIN {X 0,Y 368.535,Z 421.142,A -85,B 0,C 180,E1 -12717.238,E2 -12717.238} C_VEL
LIN {X 0,Y 368.802,Z 417.462,A -85,B 0,C 180,E1 -12719.7,E2 -12719.7} C_VEL
LIN {X 0,Y 369.283,Z 411.957,A -85,B 0,C 180,E1 -12723.498,E2 -12723.498} C_VEL
LIN {X 0,Y 369.709,Z 407.086,A -85,B 0,C 180,E1 -12727.022,E2 -12727.022} C_VEL
LIN {X 0,Y 369.782,Z 404.648,A -85,B 0,C 180,E1 -12728.843,E2 -12728.843} C_VEL
LIN {X 0,Y 369.514,Z 400.99,A -85,B 0,C 180,E1 -12731.735,E2 -12731.735} C_VEL
LIN {X 0,Y 368.946,Z 397.157,A -85,B 0,C 180,E1 -12735.043,E2 -12735.043} C_VEL
LIN {X 0,Y 368.911,Z 397.161,A -85,B 0,C 180,E1 -12738.181,E2 -12738.181} C_VEL
LIN {X 0,Y 368.915,Z 397.159,A -85,B 0,C 180,E1 -12741.359,E2 -12741.359} C_VEL
LIN {X 0,Y 368.938,Z 397.154,A -85,B 0,C 180,E1 -12745.147,E2 -12745.147} C_VEL
LIN {X 0,Y 368.93,Z 397.158,A -85,B 0,C 180,E1 -12749.047,E2 -12749.047} C_VEL
LIN {X 0,Y 368.964,Z 397.152,A -85,B 0,C 180,E1 -12752.797,E2 -12752.797} C_VEL
LIN {X 0,Y 368.938,Z 397.154,A -85,B 0,C 180,E1 -12756.116,E2 -12756.116} C_VEL
LIN {X 0,Y 368.938,Z 397.153,A -85,B 0,C 180,E1 -12759.947,E2 -12759.947} C_VEL
LIN {X 0,Y 368.981,Z 397.148,A -85,B 0,C 180,E1 -12763.399,E2 -12763.399} C_VEL
LIN {X 0,Y 369.059,Z 397.139,A -85,B 0,C 180,E1 -12766.79,E2 -12766.79} C_VEL
LIN {X 0,Y 369.069,Z 397.137,A -85,B 0,C 180,E1 -12770.132,E2 -12770.132} C_VEL
LIN {X 0,Y 369.189,Z 397.118,A -85,B 0,C 180,E1 -12772.342,E2 -12772.342} C_VEL
LIN {X 0,Y 369.146,Z 397.127,A -85,B 0,C 180,E1 -12774.538,E2 -12774.538} C_VEL
LIN {X 0,Y 369.321,Z 397.105,A -85,B 0,C 180,E1 -12777.819,E2 -12777.819} C_VEL
LIN {X 0,Y 369.46,Z 397.09,A -85,B 0,C 180,E1 -12780,E2 -12780} C_VEL
LIN {X 0,Y 369.318,Z 397.105,A -85,B 0,C 180,E1 -12782.181,E2 -12782.181} C_VEL
LIN {X 0,Y 369.205,Z 397.121,A -85,B 0,C 180,E1 -12786.626,E2 -12786.626} C_VEL
LIN {X 0,Y 369.14,Z 397.127,A -85,B 0,C 180,E1 -12788.761,E2 -12788.761} C_VEL
LIN {X 0,Y 369.007,Z 397.144,A -85,B 0,C 180,E1 -12792.093,E2 -12792.093} C_VEL
LIN {X 0,Y 369.003,Z 397.145,A -85,B 0,C 180,E1 -12795.465,E2 -12795.465} C_VEL
LIN {X 0,Y 368.984,Z 397.147,A -85,B 0,C 180,E1 -12798.893,E2 -12798.893} C_VEL
LIN {X 0,Y 368.934,Z 397.155,A -85,B 0,C 180,E1 -12802.395,E2 -12802.395} C_VEL
LIN {X 0,Y 369.001,Z 397.148,A -85,B 0,C 180,E1 -12805.98,E2 -12805.98} C_VEL
LIN {X 0,Y 368.916,Z 397.156,A -85,B 0,C 180,E1 -12809.69,E2 -12809.69} C_VEL
LIN {X 0,Y 368.9,Z 397.158,A -85,B 0,C 180,E1 -12813.044,E2 -12813.044} C_VEL
LIN {X 0,Y 368.92,Z 397.156,A -85,B 0,C 180,E1 -12816.197,E2 -12816.197} C_VEL
LIN {X 0,Y 368.906,Z 397.16,A -85,B 0,C 180,E1 -12818.953,E2 -12818.953} C_VEL
LIN {X 0,Y 368.883,Z 397.163,A -85,B 0,C 180,E1 -12822.01,E2 -12822.01} C_VEL
LIN {X 0,Y 368.909,Z 397.16,A -85,B 0,C 180,E1 -12825.18,E2 -12825.18} C_VEL
LIN {X 0,Y 368.888,Z 397.162,A -85,B 0,C 180,E1 -12826.696,E2 -12826.696} C_VEL
LIN {X 0,Y 369.008,Z 398.014,A -85,B 0,C 180,E1 -12828.195,E2 -12828.195} C_VEL
LIN {X 0,Y 369.264,Z 401.237,A -85,B 0,C 180,E1 -12831.092,E2 -12831.092} C_VEL
LIN {X 0,Y 369.198,Z 404.436,A -85,B 0,C 180,E1 -12833.835,E2 -12833.835} C_VEL
LIN {X 0,Y 368.98,Z 408.235,A -85,B 0,C 180,E1 -12836.938,E2 -12836.938} C_VEL
LIN {X 0,Y 368.628,Z 412.453,A -85,B 0,C 180,E1 -12840.284,E2 -12840.284} C_VEL
LIN {X 0,Y 368.363,Z 417.234,A -85,B 0,C 180,E1 -12843.972,E2 -12843.972} C_VEL
LIN {X 0,Y 368.176,Z 420.152,A -85,B 0,C 180,E1 -12846.152,E2 -12846.152} C_VEL
LIN {X 0,Y 372.809,Z 436.102,A -85,B 0,C 180,E1 -12846.997,E2 -12846.997} C_VEL
LIN {X 0,Y 375.898,Z 449.576,A -85,B 0,C 180,E1 -12847.865,E2 -12847.865} C_VEL
LIN {X 0,Y 377.33,Z 458.189,A -85,B 0,C 180,E1 -12848.498,E2 -12848.498} C_VEL
LIN {X 0,Y 376.314,Z 470.087,A -85,B 0,C 180,E1 -12849.359,E2 -12849.359} C_VEL
LIN {X 0,Y 375.052,Z 481.966,A -85,B 0,C 180,E1 -12850.43,E2 -12850.43} C_VEL
LIN {X 0,Y 373.694,Z 492.93,A -85,B 0,C 180,E1 -12851.638,E2 -12851.638} C_VEL
LIN {X 0,Y 372.436,Z 503.064,A -85,B 0,C 180,E1 -12852.993,E2 -12852.993} C_VEL
LIN {X 0,Y 371.108,Z 513.122,A -85,B 0,C 180,E1 -12854.625,E2 -12854.625} C_VEL
LIN {X 0,Y 370.175,Z 521.471,A -85,B 0,C 180,E1 -12856.272,E2 -12856.272} C_VEL
LIN {X 0,Y 369.094,Z 529.447,A -85,B 0,C 180,E1 -12858.189,E2 -12858.189} C_VEL
LIN {X 0,Y 368.411,Z 535.866,A -85,B 0,C 180,E1 -12860.114,E2 -12860.114} C_VEL
LIN {X 0,Y 367.847,Z 541.558,A -85,B 0,C 180,E1 -12862.314,E2 -12862.314} C_VEL
LIN {X 0,Y 367.699,Z 544.303,A -85,B 0,C 180,E1 -12863.67,E2 -12863.67} C_VEL
LIN {X 0,Y 367.509,Z 547.221,A -85,B 0,C 180,E1 -12865.613,E2 -12865.613} C_VEL
LIN {X 0,Y 367.358,Z 549.245,A -85,B 0,C 180,E1 -12867.807,E2 -12867.807} C_VEL
LIN {X 0,Y 367.373,Z 549.939,A -85,B 0,C 180,E1 -12870,E2 -12870} C_VEL
LIN {X 0,Y 367.357,Z 549.311,A -85,B 0,C 180,E1 -12872.193,E2 -12872.193} C_VEL
LIN {X 0,Y 367.507,Z 547.346,A -85,B 0,C 180,E1 -12874.387,E2 -12874.387} C_VEL
LIN {X 0,Y 367.695,Z 543.999,A -85,B 0,C 180,E1 -12876.585,E2 -12876.585} C_VEL
LIN {X 0,Y 368.06,Z 539.172,A -85,B 0,C 180,E1 -12878.787,E2 -12878.787} C_VEL
LIN {X 0,Y 368.732,Z 532.708,A -85,B 0,C 180,E1 -12880.988,E2 -12880.988} C_VEL
LIN {X 0,Y 369.661,Z 525.509,A -85,B 0,C 180,E1 -12882.908,E2 -12882.908} C_VEL
LIN {X 0,Y 370.71,Z 516.808,A -85,B 0,C 180,E1 -12884.789,E2 -12884.789} C_VEL
LIN {X 0,Y 371.897,Z 507.25,A -85,B 0,C 180,E1 -12886.467,E2 -12886.467} C_VEL
LIN {X 0,Y 373.262,Z 496.888,A -85,B 0,C 180,E1 -12887.958,E2 -12887.958} C_VEL
LIN {X 0,Y 374.67,Z 485.452,A -85,B 0,C 180,E1 -12889.306,E2 -12889.306} C_VEL
LIN {X 0,Y 376.043,Z 472.776,A -85,B 0,C 180,E1 -12890.514,E2 -12890.514} C_VEL
LIN {X 0,Y 377.148,Z 460.334,A -85,B 0,C 180,E1 -12891.459,E2 -12891.459} C_VEL
LIN {X 0,Y 377.184,Z 456.316,A -85,B 0,C 180,E1 -12891.739,E2 -12891.739} C_VEL
LIN {X 0,Y 374.421,Z 442.804,A -85,B 0,C 180,E1 -12892.695,E2 -12892.695} C_VEL
LIN {X 0,Y 370.966,Z 429.633,A -85,B 0,C 180,E1 -12893.475,E2 -12893.475} C_VEL
LIN {X 0,Y 368.159,Z 420.128,A -85,B 0,C 180,E1 -12893.971,E2 -12893.971} C_VEL
LIN {X 0,Y 368.416,Z 415.772,A -85,B 0,C 180,E1 -12897.25,E2 -12897.25} C_VEL
LIN {X 0,Y 367.808,Z 414.685,A -85,B 0,C 180,E1 -12898.149,E2 -12898.149} C_VEL
LIN {X 0,Y 365.092,Z 413.142,A -85,B 0,C 180,E1 -12899.62,E2 -12899.62} C_VEL
LIN {X 0,Y 362.801,Z 411.942,A -85,B 0,C 180,E1 -12900.811,E2 -12900.811} C_VEL
LIN {X 0,Y 361.853,Z 410.935,A -85,B 0,C 180,E1 -12901.728,E2 -12901.728} C_VEL
LIN {X 0,Y 361.794,Z 410.561,A -85,B 0,C 180,E1 -12902.036,E2 -12902.036} C_VEL
LIN {X 0,Y 362.122,Z 406.219,A -85,B 0,C 180,E1 -12905.608,E2 -12905.608} C_VEL
LIN {X 0,Y 362.229,Z 402.995,A -85,B 0,C 180,E1 -12908.38,E2 -12908.38} C_VEL
LIN {X 0,Y 362.089,Z 399.8,A -85,B 0,C 180,E1 -12911.294,E2 -12911.294} C_VEL
LIN {X 0,Y 361.888,Z 398.185,A -85,B 0,C 180,E1 -12912.821,E2 -12912.821} C_VEL
LIN {X 0,Y 361.823,Z 398.044,A -85,B 0,C 180,E1 -12915.946,E2 -12915.946} C_VEL
LIN {X 0,Y 361.838,Z 398.041,A -85,B 0,C 180,E1 -12919.245,E2 -12919.245} C_VEL
LIN {X 0,Y 361.867,Z 398.037,A -85,B 0,C 180,E1 -12922.777,E2 -12922.777} C_VEL
LIN {X 0,Y 361.858,Z 398.036,A -85,B 0,C 180,E1 -12925.72,E2 -12925.72} C_VEL
LIN {X 0,Y 361.877,Z 398.033,A -85,B 0,C 180,E1 -12929.672,E2 -12929.672} C_VEL
LIN {X 0,Y 361.956,Z 398.023,A -85,B 0,C 180,E1 -12933.475,E2 -12933.475} C_VEL
LIN {X 0,Y 361.893,Z 398.03,A -85,B 0,C 180,E1 -12937.145,E2 -12937.145} C_VEL
LIN {X 0,Y 361.923,Z 398.029,A -85,B 0,C 180,E1 -12940.724,E2 -12940.724} C_VEL
LIN {X 0,Y 361.949,Z 398.024,A -85,B 0,C 180,E1 -12944.226,E2 -12944.226} C_VEL
LIN {X 0,Y 362.002,Z 398.017,A -85,B 0,C 180,E1 -12946.528,E2 -12946.528} C_VEL
LIN {X 0,Y 362.034,Z 398.014,A -85,B 0,C 180,E1 -12949.938,E2 -12949.938} C_VEL
LIN {X 0,Y 362.154,Z 398,A -85,B 0,C 180,E1 -12952.193,E2 -12952.193} C_VEL
LIN {X 0,Y 362.121,Z 398.002,A -85,B 0,C 180,E1 -12954.431,E2 -12954.431} C_VEL
LIN {X 0,Y 362.283,Z 397.982,A -85,B 0,C 180,E1 -12957.776,E2 -12957.776} C_VEL
LIN {X 0,Y 362.429,Z 397.967,A -85,B 0,C 180,E1 -12960,E2 -12960} C_VEL
LIN {X 0,Y 362.286,Z 397.982,A -85,B 0,C 180,E1 -12962.223,E2 -12962.223} C_VEL
LIN {X 0,Y 362.175,Z 397.998,A -85,B 0,C 180,E1 -12966.686,E2 -12966.686} C_VEL
LIN {X 0,Y 362.078,Z 398.008,A -85,B 0,C 180,E1 -12968.933,E2 -12968.933} C_VEL
LIN {X 0,Y 361.963,Z 398.021,A -85,B 0,C 180,E1 -12972.332,E2 -12972.332} C_VEL
LIN {X 0,Y 361.965,Z 398.024,A -85,B 0,C 180,E1 -12974.62,E2 -12974.62} C_VEL
LIN {X 0,Y 361.962,Z 398.024,A -85,B 0,C 180,E1 -12978.099,E2 -12978.099} C_VEL
LIN {X 0,Y 361.894,Z 398.031,A -85,B 0,C 180,E1 -12981.653,E2 -12981.653} C_VEL
LIN {X 0,Y 361.931,Z 398.025,A -85,B 0,C 180,E1 -12985.29,E2 -12985.29} C_VEL
LIN {X 0,Y 361.91,Z 398.028,A -85,B 0,C 180,E1 -12987.779,E2 -12987.779} C_VEL
LIN {X 0,Y 361.839,Z 398.038,A -85,B 0,C 180,E1 -12991.629,E2 -12991.629} C_VEL
LIN {X 0,Y 361.877,Z 398.036,A -85,B 0,C 180,E1 -12995.345,E2 -12995.345} C_VEL
LIN {X 0,Y 361.877,Z 398.039,A -85,B 0,C 180,E1 -12999.028,E2 -12999.028} C_VEL
LIN {X 0,Y 361.858,Z 398.039,A -85,B 0,C 180,E1 -13002.435,E2 -13002.435} C_VEL
LIN {X 0,Y 361.898,Z 398.119,A -85,B 0,C 180,E1 -13004.746,E2 -13004.746} C_VEL
LIN {X 0,Y 362.59,Z 402.793,A -85,B 0,C 180,E1 -13008.775,E2 -13008.775} C_VEL
LIN {X 0,Y 362.712,Z 406.455,A -85,B 0,C 180,E1 -13011.681,E2 -13011.681} C_VEL
LIN {X 0,Y 362.5,Z 410.229,A -85,B 0,C 180,E1 -13014.516,E2 -13014.516} C_VEL
LIN {X 0,Y 362.161,Z 413.76,A -85,B 0,C 180,E1 -13017.087,E2 -13017.087} C_VEL
LIN {X 0,Y 361.691,Z 419.317,A -85,B 0,C 180,E1 -13020.973,E2 -13020.973} C_VEL
LIN {X 0,Y 361.239,Z 424.76,A -85,B 0,C 180,E1 -13024.658,E2 -13024.658} C_VEL
LIN {X 0,Y 361.183,Z 426.296,A -85,B 0,C 180,E1 -13025.607,E2 -13025.607} C_VEL
LIN {X 0,Y 365.334,Z 441.041,A -85,B 0,C 180,E1 -13026.372,E2 -13026.372} C_VEL
LIN {X 0,Y 368.283,Z 454.162,A -85,B 0,C 180,E1 -13027.205,E2 -13027.205} C_VEL
LIN {X 0,Y 370.354,Z 466.572,A -85,B 0,C 180,E1 -13028.136,E2 -13028.136} C_VEL
LIN {X 0,Y 369.161,Z 479.447,A -85,B 0,C 180,E1 -13029.123,E2 -13029.123} C_VEL
LIN {X 0,Y 367.7,Z 491.837,A -85,B 0,C 180,E1 -13030.313,E2 -13030.313} C_VEL
LIN {X 0,Y 366.229,Z 503.369,A -85,B 0,C 180,E1 -13031.685,E2 -13031.685} C_VEL
LIN {X 0,Y 364.839,Z 513.817,A -85,B 0,C 180,E1 -13033.205,E2 -13033.205} C_VEL
LIN {X 0,Y 363.554,Z 523.546,A -85,B 0,C 180,E1 -13034.929,E2 -13034.929} C_VEL
LIN {X 0,Y 362.522,Z 532.251,A -85,B 0,C 180,E1 -13036.833,E2 -13036.833} C_VEL
LIN {X 0,Y 361.517,Z 539.514,A -85,B 0,C 180,E1 -13038.79,E2 -13038.79} C_VEL
LIN {X 0,Y 361.02,Z 544.607,A -85,B 0,C 180,E1 -13040.475,E2 -13040.475} C_VEL
LIN {X 0,Y 360.588,Z 549.863,A -85,B 0,C 180,E1 -13042.722,E2 -13042.722} C_VEL
LIN {X 0,Y 360.394,Z 552.807,A -85,B 0,C 180,E1 -13044.404,E2 -13044.404} C_VEL
LIN {X 0,Y 360.268,Z 555.5,A -85,B 0,C 180,E1 -13046.645,E2 -13046.645} C_VEL
LIN {X 0,Y 360.246,Z 556.834,A -85,B 0,C 180,E1 -13048.882,E2 -13048.882} C_VEL
LIN {X 0,Y 360.246,Z 556.832,A -85,B 0,C 180,E1 -13051.118,E2 -13051.118} C_VEL
LIN {X 0,Y 360.268,Z 555.494,A -85,B 0,C 180,E1 -13053.355,E2 -13053.355} C_VEL
LIN {X 0,Y 360.411,Z 552.796,A -85,B 0,C 180,E1 -13055.595,E2 -13055.595} C_VEL
LIN {X 0,Y 360.66,Z 548.661,A -85,B 0,C 180,E1 -13057.84,E2 -13057.84} C_VEL
LIN {X 0,Y 361.18,Z 542.966,A -85,B 0,C 180,E1 -13060.086,E2 -13060.086} C_VEL
LIN {X 0,Y 361.939,Z 536.547,A -85,B 0,C 180,E1 -13062.048,E2 -13062.048} C_VEL
LIN {X 0,Y 362.91,Z 528.571,A -85,B 0,C 180,E1 -13064.009,E2 -13064.009} C_VEL
LIN {X 0,Y 363.975,Z 520.228,A -85,B 0,C 180,E1 -13065.684,E2 -13065.684} C_VEL
LIN {X 0,Y 365.349,Z 510.183,A -85,B 0,C 180,E1 -13067.347,E2 -13067.347} C_VEL
LIN {X 0,Y 366.82,Z 498.976,A -85,B 0,C 180,E1 -13068.863,E2 -13068.863} C_VEL
LIN {X 0,Y 368.364,Z 486.481,A -85,B 0,C 180,E1 -13070.223,E2 -13070.223} C_VEL
LIN {X 0,Y 369.654,Z 474.016,A -85,B 0,C 180,E1 -13071.313,E2 -13071.313} C_VEL
LIN {X 0,Y 370.195,Z 465.408,A -85,B 0,C 180,E1 -13071.947,E2 -13071.947} C_VEL
LIN {X 0,Y 367.825,Z 451.838,A -85,B 0,C 180,E1 -13072.944,E2 -13072.944} C_VEL
LIN {X 0,Y 364.723,Z 438.687,A -85,B 0,C 180,E1 -13073.753,E2 -13073.753} C_VEL
LIN {X 0,Y 361.179,Z 426.14,A -85,B 0,C 180,E1 -13074.408,E2 -13074.408} C_VEL
LIN {X 0,Y 361.552,Z 421.065,A -85,B 0,C 180,E1 -13077.809,E2 -13077.809} C_VEL
LIN {X 0,Y 361.982,Z 415.563,A -85,B 0,C 180,E1 -13081.615,E2 -13081.615} C_VEL
LIN {X 0,Y 362.337,Z 411.917,A -85,B 0,C 180,E1 -13084.228,E2 -13084.228} C_VEL
LIN {X 0,Y 362.685,Z 407.628,A -85,B 0,C 180,E1 -13087.393,E2 -13087.393} C_VEL
LIN {X 0,Y 362.695,Z 404.592,A -85,B 0,C 180,E1 -13089.751,E2 -13089.751} C_VEL
LIN {X 0,Y 362.34,Z 401.232,A -85,B 0,C 180,E1 -13092.519,E2 -13092.519} C_VEL
LIN {X 0,Y 361.872,Z 398.038,A -85,B 0,C 180,E1 -13095.445,E2 -13095.445} C_VEL
LIN {X 0,Y 361.873,Z 398.037,A -85,B 0,C 180,E1 -13099.238,E2 -13099.238} C_VEL
LIN {X 0,Y 361.875,Z 398.036,A -85,B 0,C 180,E1 -13102.983,E2 -13102.983} C_VEL
LIN {X 0,Y 361.861,Z 398.036,A -85,B 0,C 180,E1 -13106.63,E2 -13106.63} C_VEL
LIN {X 0,Y 361.873,Z 398.035,A -85,B 0,C 180,E1 -13109.672,E2 -13109.672} C_VEL
LIN {X 0,Y 361.955,Z 398.024,A -85,B 0,C 180,E1 -13113.475,E2 -13113.475} C_VEL
LIN {X 0,Y 361.883,Z 398.034,A -85,B 0,C 180,E1 -13117.144,E2 -13117.144} C_VEL
LIN {X 0,Y 361.922,Z 398.029,A -85,B 0,C 180,E1 -13120.724,E2 -13120.724} C_VEL
LIN {X 0,Y 361.95,Z 398.024,A -85,B 0,C 180,E1 -13124.226,E2 -13124.226} C_VEL
LIN {X 0,Y 362,Z 398.016,A -85,B 0,C 180,E1 -13126.528,E2 -13126.528} C_VEL
LIN {X 0,Y 362.033,Z 398.012,A -85,B 0,C 180,E1 -13129.938,E2 -13129.938} C_VEL
LIN {X 0,Y 362.153,Z 397.995,A -85,B 0,C 180,E1 -13132.193,E2 -13132.193} C_VEL
LIN {X 0,Y 362.12,Z 398.002,A -85,B 0,C 180,E1 -13134.431,E2 -13134.431} C_VEL
LIN {X 0,Y 362.284,Z 397.981,A -85,B 0,C 180,E1 -13137.777,E2 -13137.777} C_VEL
LIN {X 0,Y 362.43,Z 397.966,A -85,B 0,C 180,E1 -13140,E2 -13140} C_VEL
LIN {X 0,Y 362.282,Z 397.981,A -85,B 0,C 180,E1 -13142.224,E2 -13142.224} C_VEL
LIN {X 0,Y 362.174,Z 397.998,A -85,B 0,C 180,E1 -13146.686,E2 -13146.686} C_VEL
LIN {X 0,Y 362.076,Z 398.007,A -85,B 0,C 180,E1 -13148.933,E2 -13148.933} C_VEL
LIN {X 0,Y 361.962,Z 398.022,A -85,B 0,C 180,E1 -13152.332,E2 -13152.332} C_VEL
LIN {X 0,Y 361.965,Z 398.022,A -85,B 0,C 180,E1 -13154.62,E2 -13154.62} C_VEL
LIN {X 0,Y 361.961,Z 398.024,A -85,B 0,C 180,E1 -13158.099,E2 -13158.099} C_VEL
LIN {X 0,Y 361.893,Z 398.031,A -85,B 0,C 180,E1 -13161.653,E2 -13161.653} C_VEL
LIN {X 0,Y 361.93,Z 398.026,A -85,B 0,C 180,E1 -13165.29,E2 -13165.29} C_VEL
LIN {X 0,Y 361.91,Z 398.031,A -85,B 0,C 180,E1 -13167.779,E2 -13167.779} C_VEL
LIN {X 0,Y 361.839,Z 398.038,A -85,B 0,C 180,E1 -13171.629,E2 -13171.629} C_VEL
LIN {X 0,Y 361.876,Z 398.034,A -85,B 0,C 180,E1 -13175.345,E2 -13175.345} C_VEL
LIN {X 0,Y 361.873,Z 398.037,A -85,B 0,C 180,E1 -13179.027,E2 -13179.027} C_VEL
LIN {X 0,Y 361.838,Z 398.039,A -85,B 0,C 180,E1 -13182.829,E2 -13182.829} C_VEL
LIN {X 0,Y 361.831,Z 398.04,A -85,B 0,C 180,E1 -13185.945,E2 -13185.945} C_VEL
LIN {X 0,Y 361.85,Z 398.061,A -85,B 0,C 180,E1 -13187.173,E2 -13187.173} C_VEL
LIN {X 0,Y 362.201,Z 401.277,A -85,B 0,C 180,E1 -13190.184,E2 -13190.184} C_VEL
LIN {X 0,Y 362.241,Z 404.505,A -85,B 0,C 180,E1 -13193.027,E2 -13193.027} C_VEL
LIN {X 0,Y 361.961,Z 408.753,A -85,B 0,C 180,E1 -13196.606,E2 -13196.606} C_VEL
LIN {X 0,Y 361.648,Z 412.515,A -85,B 0,C 180,E1 -13199.651,E2 -13199.651} C_VEL
LIN {X 0,Y 361.336,Z 417.367,A -85,B 0,C 180,E1 -13203.471,E2 -13203.471} C_VEL
LIN {X 0,Y 361.14,Z 420.204,A -85,B 0,C 180,E1 -13205.65,E2 -13205.65} C_VEL
LIN {X 0,Y 365.845,Z 436.202,A -85,B 0,C 180,E1 -13206.533,E2 -13206.533} C_VEL
LIN {X 0,Y 368.73,Z 448.351,A -85,B 0,C 180,E1 -13207.337,E2 -13207.337} C_VEL
LIN {X 0,Y 370.602,Z 458.654,A -85,B 0,C 180,E1 -13208.117,E2 -13208.117} C_VEL
LIN {X 0,Y 369.499,Z 471.742,A -85,B 0,C 180,E1 -13209.107,E2 -13209.107} C_VEL
LIN {X 0,Y 368.042,Z 484.618,A -85,B 0,C 180,E1 -13210.333,E2 -13210.333} C_VEL
LIN {X 0,Y 366.477,Z 496.206,A -85,B 0,C 180,E1 -13211.698,E2 -13211.698} C_VEL
LIN {X 0,Y 365.122,Z 506.694,A -85,B 0,C 180,E1 -13213.218,E2 -13213.218} C_VEL
LIN {X 0,Y 363.733,Z 516.952,A -85,B 0,C 180,E1 -13215.038,E2 -13215.038} C_VEL
LIN {X 0,Y 362.771,Z 525.185,A -85,B 0,C 180,E1 -13216.842,E2 -13216.842} C_VEL
LIN {X 0,Y 361.754,Z 532.456,A -85,B 0,C 180,E1 -13218.798,E2 -13218.798} C_VEL
LIN {X 0,Y 361.207,Z 537.544,A -85,B 0,C 180,E1 -13220.481,E2 -13220.481} C_VEL
LIN {X 0,Y 360.704,Z 542.821,A -85,B 0,C 180,E1 -13222.724,E2 -13222.724} C_VEL
LIN {X 0,Y 360.498,Z 545.765,A -85,B 0,C 180,E1 -13224.406,E2 -13224.406} C_VEL
LIN {X 0,Y 360.308,Z 548.471,A -85,B 0,C 180,E1 -13226.645,E2 -13226.645} C_VEL
LIN {X 0,Y 360.257,Z 549.826,A -85,B 0,C 180,E1 -13228.882,E2 -13228.882} C_VEL
LIN {X 0,Y 360.257,Z 549.859,A -85,B 0,C 180,E1 -13231.118,E2 -13231.118} C_VEL
LIN {X 0,Y 360.307,Z 548.567,A -85,B 0,C 180,E1 -13233.355,E2 -13233.355} C_VEL
LIN {X 0,Y 360.496,Z 545.919,A -85,B 0,C 180,E1 -13235.594,E2 -13235.594} C_VEL
LIN {X 0,Y 360.774,Z 541.848,A -85,B 0,C 180,E1 -13237.838,E2 -13237.838} C_VEL
LIN {X 0,Y 361.339,Z 536.223,A -85,B 0,C 180,E1 -13240.082,E2 -13240.082} C_VEL
LIN {X 0,Y 362.067,Z 529.873,A -85,B 0,C 180,E1 -13242.044,E2 -13242.044} C_VEL
LIN {X 0,Y 363.184,Z 521.975,A -85,B 0,C 180,E1 -13243.998,E2 -13243.998} C_VEL
LIN {X 0,Y 364.211,Z 513.714,A -85,B 0,C 180,E1 -13245.673,E2 -13245.673} C_VEL
LIN {X 0,Y 365.575,Z 503.759,A -85,B 0,C 180,E1 -13247.336,E2 -13247.336} C_VEL
LIN {X 0,Y 367.052,Z 492.677,A -85,B 0,C 180,E1 -13248.851,E2 -13248.851} C_VEL
LIN {X 0,Y 368.574,Z 480.24,A -85,B 0,C 180,E1 -13250.219,E2 -13250.219} C_VEL
LIN {X 0,Y 369.896,Z 468.153,A -85,B 0,C 180,E1 -13251.288,E2 -13251.288} C_VEL
LIN {X 0,Y 370.631,Z 458.311,A -85,B 0,C 180,E1 -13252.009,E2 -13252.009} C_VEL
LIN {X 0,Y 368.058,Z 445.305,A -85,B 0,C 180,E1 -13252.985,E2 -13252.985} C_VEL
LIN {X 0,Y 364.549,Z 431.65,A -85,B 0,C 180,E1 -13253.847,E2 -13253.847} C_VEL
LIN {X 0,Y 361.132,Z 420.213,A -85,B 0,C 180,E1 -13254.449,E2 -13254.449} C_VEL
LIN {X 0,Y 361.417,Z 415.849,A -85,B 0,C 180,E1 -13257.82,E2 -13257.82} C_VEL
LIN {X 0,Y 361.776,Z 411.057,A -85,B 0,C 180,E1 -13261.636,E2 -13261.636} C_VEL
LIN {X 0,Y 361.794,Z 410.561,A -85,B 0,C 180,E1 -13262.036,E2 -13262.036} C_VEL
LIN {X 0,Y 361.208,Z 409.52,A -85,B 0,C 180,E1 -13262.952,E2 -13262.952} C_VEL
LIN {X 0,Y 358.504,Z 408.078,A -85,B 0,C 180,E1 -13264.454,E2 -13264.454} C_VEL
LIN {X 0,Y 356.194,Z 406.97,A -85,B 0,C 180,E1 -13265.669,E2 -13265.669} C_VEL
LIN {X 0,Y 355.214,Z 406.033,A -85,B 0,C 180,E1 -13266.605,E2 -13266.605} C_VEL
LIN {X 0,Y 355.142,Z 405.684,A -85,B 0,C 180,E1 -13266.92,E2 -13266.92} C_VEL
LIN {X 0,Y 355.193,Z 402.831,A -85,B 0,C 180,E1 -13269.496,E2 -13269.496} C_VEL
LIN {X 0,Y 354.959,Z 399.841,A -85,B 0,C 180,E1 -13272.313,E2 -13272.313} C_VEL
LIN {X 0,Y 354.887,Z 399.255,A -85,B 0,C 180,E1 -13272.884,E2 -13272.884} C_VEL
LIN {X 0,Y 354.826,Z 398.917,A -85,B 0,C 180,E1 -13274.516,E2 -13274.516} C_VEL
LIN {X 0,Y 354.797,Z 398.921,A -85,B 0,C 180,E1 -13277.663,E2 -13277.663} C_VEL
LIN {X 0,Y 354.817,Z 398.914,A -85,B 0,C 180,E1 -13280.666,E2 -13280.666} C_VEL
LIN {X 0,Y 354.825,Z 398.913,A -85,B 0,C 180,E1 -13284.301,E2 -13284.301} C_VEL
LIN {X 0,Y 354.79,Z 398.916,A -85,B 0,C 180,E1 -13287.667,E2 -13287.667} C_VEL
LIN {X 0,Y 354.871,Z 398.905,A -85,B 0,C 180,E1 -13290.621,E2 -13290.621} C_VEL
LIN {X 0,Y 354.902,Z 398.904,A -85,B 0,C 180,E1 -13294.173,E2 -13294.173} C_VEL
LIN {X 0,Y 354.837,Z 398.91,A -85,B 0,C 180,E1 -13297.894,E2 -13297.894} C_VEL
LIN {X 0,Y 354.926,Z 398.9,A -85,B 0,C 180,E1 -13301.891,E2 -13301.891} C_VEL
LIN {X 0,Y 354.945,Z 398.896,A -85,B 0,C 180,E1 -13305.981,E2 -13305.981} C_VEL
LIN {X 0,Y 354.981,Z 398.892,A -85,B 0,C 180,E1 -13309.736,E2 -13309.736} C_VEL
LIN {X 0,Y 355.117,Z 398.878,A -85,B 0,C 180,E1 -13312.037,E2 -13312.037} C_VEL
LIN {X 0,Y 355.095,Z 398.877,A -85,B 0,C 180,E1 -13314.321,E2 -13314.321} C_VEL
LIN {X 0,Y 355.247,Z 398.858,A -85,B 0,C 180,E1 -13317.732,E2 -13317.732} C_VEL
LIN {X 0,Y 355.399,Z 398.842,A -85,B 0,C 180,E1 -13320,E2 -13320} C_VEL
LIN {X 0,Y 355.249,Z 398.858,A -85,B 0,C 180,E1 -13322.268,E2 -13322.268} C_VEL
LIN {X 0,Y 355.141,Z 398.873,A -85,B 0,C 180,E1 -13326.819,E2 -13326.819} C_VEL
LIN {X 0,Y 355.019,Z 398.887,A -85,B 0,C 180,E1 -13329.112,E2 -13329.112} C_VEL
LIN {X 0,Y 354.924,Z 398.899,A -85,B 0,C 180,E1 -13332.581,E2 -13332.581} C_VEL
LIN {X 0,Y 354.892,Z 398.905,A -85,B 0,C 180,E1 -13336.096,E2 -13336.096} C_VEL
LIN {X 0,Y 354.909,Z 398.9,A -85,B 0,C 180,E1 -13338.472,E2 -13338.472} C_VEL
LIN {X 0,Y 354.837,Z 398.91,A -85,B 0,C 180,E1 -13342.106,E2 -13342.106} C_VEL
LIN {X 0,Y 354.901,Z 398.904,A -85,B 0,C 180,E1 -13345.827,E2 -13345.827} C_VEL
LIN {X 0,Y 354.819,Z 398.909,A -85,B 0,C 180,E1 -13349.682,E2 -13349.682} C_VEL
LIN {X 0,Y 354.808,Z 398.916,A -85,B 0,C 180,E1 -13353.702,E2 -13353.702} C_VEL
LIN {X 0,Y 354.804,Z 398.917,A -85,B 0,C 180,E1 -13356.459,E2 -13356.459} C_VEL
LIN {X 0,Y 354.826,Z 398.916,A -85,B 0,C 180,E1 -13359.423,E2 -13359.423} C_VEL
LIN {X 0,Y 354.807,Z 398.917,A -85,B 0,C 180,E1 -13362.87,E2 -13362.87} C_VEL
LIN {X 0,Y 354.861,Z 399.116,A -85,B 0,C 180,E1 -13364.522,E2 -13364.522} C_VEL
LIN {X 0,Y 355.388,Z 402.751,A -85,B 0,C 180,E1 -13367.75,E2 -13367.75} C_VEL
LIN {X 0,Y 355.717,Z 405.912,A -85,B 0,C 180,E1 -13370.402,E2 -13370.402} C_VEL
LIN {X 0,Y 355.678,Z 408.228,A -85,B 0,C 180,E1 -13372.226,E2 -13372.226} C_VEL
LIN {X 0,Y 355.386,Z 411.879,A -85,B 0,C 180,E1 -13375.005,E2 -13375.005} C_VEL
LIN {X 0,Y 354.937,Z 416.473,A -85,B 0,C 180,E1 -13378.368,E2 -13378.368} C_VEL
LIN {X 0,Y 354.543,Z 421.025,A -85,B 0,C 180,E1 -13381.592,E2 -13381.592} C_VEL
LIN {X 0,Y 354.166,Z 426.103,A -85,B 0,C 180,E1 -13385.087,E2 -13385.087} C_VEL
LIN {X 0,Y 356.935,Z 435.674,A -85,B 0,C 180,E1 -13385.576,E2 -13385.576} C_VEL
LIN {X 0,Y 360.411,Z 449.414,A -85,B 0,C 180,E1 -13386.419,E2 -13386.419} C_VEL
LIN {X 0,Y 362.869,Z 462.314,A -85,B 0,C 180,E1 -13387.36,E2 -13387.36} C_VEL
LIN {X 0,Y 363.629,Z 468.499,A -85,B 0,C 180,E1 -13387.86,E2 -13387.86} C_VEL
LIN {X 0,Y 362.303,Z 481.381,A -85,B 0,C 180,E1 -13388.897,E2 -13388.897} C_VEL
LIN {X 0,Y 360.836,Z 493.064,A -85,B 0,C 180,E1 -13390.071,E2 -13390.071} C_VEL
LIN {X 0,Y 359.319,Z 504.368,A -85,B 0,C 180,E1 -13391.468,E2 -13391.468} C_VEL
LIN {X 0,Y 357.762,Z 515.437,A -85,B 0,C 180,E1 -13393.157,E2 -13393.157} C_VEL
LIN {X 0,Y 356.489,Z 524.571,A -85,B 0,C 180,E1 -13394.858,E2 -13394.858} C_VEL
LIN {X 0,Y 355.424,Z 533.301,A -85,B 0,C 180,E1 -13396.856,E2 -13396.856} C_VEL
LIN {X 0,Y 354.509,Z 539.446,A -85,B 0,C 180,E1 -13398.565,E2 -13398.565} C_VEL
LIN {X 0,Y 353.987,Z 544.539,A -85,B 0,C 180,E1 -13400.284,E2 -13400.284} C_VEL
LIN {X 0,Y 353.51,Z 549.795,A -85,B 0,C 180,E1 -13402.575,E2 -13402.575} C_VEL
LIN {X 0,Y 353.329,Z 552.739,A -85,B 0,C 180,E1 -13404.292,E2 -13404.292} C_VEL
LIN {X 0,Y 353.191,Z 555.432,A -85,B 0,C 180,E1 -13406.578,E2 -13406.578} C_VEL
LIN {X 0,Y 353.146,Z 556.765,A -85,B 0,C 180,E1 -13408.86,E2 -13408.86} C_VEL
LIN {X 0,Y 353.146,Z 556.763,A -85,B 0,C 180,E1 -13411.14,E2 -13411.14} C_VEL
LIN {X 0,Y 353.192,Z 555.425,A -85,B 0,C 180,E1 -13413.422,E2 -13413.422} C_VEL
LIN {X 0,Y 353.329,Z 552.727,A -85,B 0,C 180,E1 -13415.708,E2 -13415.708} C_VEL
LIN {X 0,Y 353.604,Z 548.591,A -85,B 0,C 180,E1 -13417.997,E2 -13417.997} C_VEL
LIN {X 0,Y 354.161,Z 542.896,A -85,B 0,C 180,E1 -13420.288,E2 -13420.288} C_VEL
LIN {X 0,Y 354.966,Z 536.476,A -85,B 0,C 180,E1 -13422.289,E2 -13422.289} C_VEL
LIN {X 0,Y 355.956,Z 528.744,A -85,B 0,C 180,E1 -13424.231,E2 -13424.231} C_VEL
LIN {X 0,Y 357.085,Z 520.156,A -85,B 0,C 180,E1 -13425.994,E2 -13425.994} C_VEL
LIN {X 0,Y 358.518,Z 510.111,A -85,B 0,C 180,E1 -13427.689,E2 -13427.689} C_VEL
LIN {X 0,Y 360.057,Z 498.903,A -85,B 0,C 180,E1 -13429.231,E2 -13429.231} C_VEL
LIN {X 0,Y 361.681,Z 486.509,A -85,B 0,C 180,E1 -13430.603,E2 -13430.603} C_VEL
LIN {X 0,Y 363.028,Z 474.017,A -85,B 0,C 180,E1 -13431.716,E2 -13431.716} C_VEL
LIN {X 0,Y 363.554,Z 468.324,A -85,B 0,C 180,E1 -13432.145,E2 -13432.145} C_VEL
LIN {X 0,Y 362.026,Z 457.549,A -85,B 0,C 180,E1 -13432.997,E2 -13432.997} C_VEL
LIN {X 0,Y 359.106,Z 443.738,A -85,B 0,C 180,E1 -13433.934,E2 -13433.934} C_VEL
LIN {X 0,Y 355.069,Z 429.435,A -85,B 0,C 180,E1 -13434.744,E2 -13434.744} C_VEL
LIN {X 0,Y 354.164,Z 426.081,A -85,B 0,C 180,E1 -13434.913,E2 -13434.913} C_VEL
LIN {X 0,Y 354.539,Z 421.002,A -85,B 0,C 180,E1 -13438.408,E2 -13438.408} C_VEL
LIN {X 0,Y 355.021,Z 415.516,A -85,B 0,C 180,E1 -13442.309,E2 -13442.309} C_VEL
LIN {X 0,Y 355.492,Z 410.706,A -85,B 0,C 180,E1 -13445.849,E2 -13445.849} C_VEL
LIN {X 0,Y 355.727,Z 406.358,A -85,B 0,C 180,E1 -13449.214,E2 -13449.214} C_VEL
LIN {X 0,Y 355.584,Z 403.807,A -85,B 0,C 180,E1 -13451.318,E2 -13451.318} C_VEL
LIN {X 0,Y 355.055,Z 400.092,A -85,B 0,C 180,E1 -13454.554,E2 -13454.554} C_VEL
LIN {X 0,Y 354.84,Z 398.914,A -85,B 0,C 180,E1 -13455.796,E2 -13455.796} C_VEL
LIN {X 0,Y 354.825,Z 398.915,A -85,B 0,C 180,E1 -13459.184,E2 -13459.184} C_VEL
LIN {X 0,Y 354.814,Z 398.915,A -85,B 0,C 180,E1 -13462.401,E2 -13462.401} C_VEL
LIN {X 0,Y 354.813,Z 398.914,A -85,B 0,C 180,E1 -13464.941,E2 -13464.941} C_VEL
LIN {X 0,Y 354.794,Z 398.917,A -85,B 0,C 180,E1 -13468.405,E2 -13468.405} C_VEL
LIN {X 0,Y 354.847,Z 398.909,A -85,B 0,C 180,E1 -13471.619,E2 -13471.619} C_VEL
LIN {X 0,Y 354.899,Z 398.904,A -85,B 0,C 180,E1 -13474.173,E2 -13474.173} C_VEL
LIN {X 0,Y 354.818,Z 398.912,A -85,B 0,C 180,E1 -13477.893,E2 -13477.893} C_VEL
LIN {X 0,Y 354.924,Z 398.899,A -85,B 0,C 180,E1 -13481.891,E2 -13481.891} C_VEL
LIN {X 0,Y 354.944,Z 398.895,A -85,B 0,C 180,E1 -13485.981,E2 -13485.981} C_VEL
LIN {X 0,Y 354.98,Z 398.889,A -85,B 0,C 180,E1 -13489.736,E2 -13489.736} C_VEL
LIN {X 0,Y 355.115,Z 398.873,A -85,B 0,C 180,E1 -13492.037,E2 -13492.037} C_VEL
LIN {X 0,Y 355.094,Z 398.877,A -85,B 0,C 180,E1 -13494.321,E2 -13494.321} C_VEL
LIN {X 0,Y 355.248,Z 398.858,A -85,B 0,C 180,E1 -13497.732,E2 -13497.732} C_VEL
LIN {X 0,Y 355.399,Z 398.841,A -85,B 0,C 180,E1 -13500,E2 -13500} C_VEL
LIN {X 0,Y 355.245,Z 398.858,A -85,B 0,C 180,E1 -13502.268,E2 -13502.268} C_VEL
LIN {X 0,Y 355.14,Z 398.873,A -85,B 0,C 180,E1 -13506.819,E2 -13506.819} C_VEL
LIN {X 0,Y 355.017,Z 398.887,A -85,B 0,C 180,E1 -13509.112,E2 -13509.112} C_VEL
